LIN {X 0,Y 573.262,Z 307.702,A -85,B 0,C 180,E1 -2310.634,E2 -2310.634} C_VEL
LIN {X 0,Y 573.263,Z 307.696,A -85,B 0,C 180,E1 -2313.5,E2 -2313.5} C_VEL
LIN {X 0,Y 573.221,Z 307.71,A -85,B 0,C 180,E1 -2316.134,E2 -2316.134} C_VEL
LIN {X 0,Y 573.242,Z 307.699,A -85,B 0,C 180,E1 -2319.173,E2 -2319.173} C_VEL
LIN {X 0,Y 573.221,Z 307.701,A -85,B 0,C 180,E1 -2321.411,E2 -2321.411} C_VEL
LIN {X 0,Y 573.236,Z 307.703,A -85,B 0,C 180,E1 -2323.621,E2 -2323.621} C_VEL
LIN {X 0,Y 573.263,Z 307.702,A -85,B 0,C 180,E1 -2325.807,E2 -2325.807} C_VEL
LIN {X 0,Y 573.254,Z 307.697,A -85,B 0,C 180,E1 -2328.745,E2 -2328.745} C_VEL
LIN {X 0,Y 573.271,Z 307.7,A -85,B 0,C 180,E1 -2331.54,E2 -2331.54} C_VEL
LIN {X 0,Y 573.231,Z 307.706,A -85,B 0,C 180,E1 -2333.665,E2 -2333.665} C_VEL
LIN {X 0,Y 573.212,Z 307.713,A -85,B 0,C 180,E1 -2335.781,E2 -2335.781} C_VEL
LIN {X 0,Y 573.289,Z 307.701,A -85,B 0,C 180,E1 -2337.892,E2 -2337.892} C_VEL
LIN {X 0,Y 573.301,Z 307.696,A -85,B 0,C 180,E1 -2340,E2 -2340} C_VEL
LIN {X 0,Y 573.272,Z 307.695,A -85,B 0,C 180,E1 -2342.811,E2 -2342.811} C_VEL
LIN {X 0,Y 573.263,Z 307.705,A -85,B 0,C 180,E1 -2345.628,E2 -2345.628} C_VEL
LIN {X 0,Y 573.22,Z 307.701,A -85,B 0,C 180,E1 -2348.46,E2 -2348.46} C_VEL
LIN {X 0,Y 573.261,Z 307.704,A -85,B 0,C 180,E1 -2351.312,E2 -2351.312} C_VEL
LIN {X 0,Y 573.214,Z 307.703,A -85,B 0,C 180,E1 -2354.402,E2 -2354.402} C_VEL
LIN {X 0,Y 573.226,Z 307.706,A -85,B 0,C 180,E1 -2357.112,E2 -2357.112} C_VEL
LIN {X 0,Y 573.217,Z 307.703,A -85,B 0,C 180,E1 -2360.078,E2 -2360.078} C_VEL
LIN {X 0,Y 573.207,Z 307.703,A -85,B 0,C 180,E1 -2362.339,E2 -2362.339} C_VEL
LIN {X 0,Y 573.184,Z 307.706,A -85,B 0,C 180,E1 -2364.34,E2 -2364.34} C_VEL
LIN {X 0,Y 572.546,Z 307.793,A -85,B 0,C 180,E1 -2364.927,E2 -2364.927} C_VEL
LIN {X 0,Y 569.716,Z 308.148,A -85,B 0,C 180,E1 -2365.879,E2 -2365.879} C_VEL
LIN {X 0,Y 567.302,Z 308.45,A -85,B 0,C 180,E1 -2366.645,E2 -2366.645} C_VEL
LIN {X 0,Y 566.251,Z 308.577,A -85,B 0,C 180,E1 -2367.236,E2 -2367.236} C_VEL
LIN {X 0,Y 566.158,Z 308.585,A -85,B 0,C 180,E1 -2367.436,E2 -2367.436} C_VEL
LIN {X 0,Y 566.159,Z 308.583,A -85,B 0,C 180,E1 -2369.771,E2 -2369.771} C_VEL
LIN {X 0,Y 566.189,Z 308.58,A -85,B 0,C 180,E1 -2372.429,E2 -2372.429} C_VEL
LIN {X 0,Y 566.168,Z 308.591,A -85,B 0,C 180,E1 -2374.989,E2 -2374.989} C_VEL
LIN {X 0,Y 566.186,Z 308.581,A -85,B 0,C 180,E1 -2377.461,E2 -2377.461} C_VEL
LIN {X 0,Y 566.197,Z 308.578,A -85,B 0,C 180,E1 -2380.199,E2 -2380.199} C_VEL
LIN {X 0,Y 566.191,Z 308.584,A -85,B 0,C 180,E1 -2383.055,E2 -2383.055} C_VEL
LIN {X 0,Y 566.185,Z 308.579,A -85,B 0,C 180,E1 -2386.05,E2 -2386.05} C_VEL
LIN {X 0,Y 566.195,Z 308.582,A -85,B 0,C 180,E1 -2389.215,E2 -2389.215} C_VEL
LIN {X 0,Y 566.227,Z 308.615,A -85,B 0,C 180,E1 -2391.146,E2 -2391.146} C_VEL
LIN {X 0,Y 566.73,Z 313.138,A -85,B 0,C 180,E1 -2391.908,E2 -2391.908} C_VEL
LIN {X 0,Y 566.547,Z 330.448,A -85,B 0,C 180,E1 -2394.685,E2 -2394.685} C_VEL
LIN {X 0,Y 566.522,Z 332.949,A -85,B 0,C 180,E1 -2395.082,E2 -2395.082} C_VEL
LIN {X 0,Y 567.796,Z 340.155,A -85,B 0,C 180,E1 -2395.217,E2 -2395.217} C_VEL
LIN {X 0,Y 567.419,Z 469.812,A -85,B 0,C 180,E1 -2396.898,E2 -2396.898} C_VEL
LIN {X 0,Y 567.292,Z 484.271,A -85,B 0,C 180,E1 -2397.238,E2 -2397.238} C_VEL
LIN {X 0,Y 567.159,Z 497.173,A -85,B 0,C 180,E1 -2397.674,E2 -2397.674} C_VEL
LIN {X 0,Y 567.003,Z 509.326,A -85,B 0,C 180,E1 -2398.212,E2 -2398.212} C_VEL
LIN {X 0,Y 566.77,Z 521.671,A -85,B 0,C 180,E1 -2398.901,E2 -2398.901} C_VEL
LIN {X 0,Y 566.622,Z 533.823,A -85,B 0,C 180,E1 -2399.744,E2 -2399.744} C_VEL
LIN {X 0,Y 566.424,Z 545.722,A -85,B 0,C 180,E1 -2400.756,E2 -2400.756} C_VEL
LIN {X 0,Y 566.262,Z 556.36,A -85,B 0,C 180,E1 -2401.861,E2 -2401.861} C_VEL
LIN {X 0,Y 566.116,Z 565.674,A -85,B 0,C 180,E1 -2403.045,E2 -2403.045} C_VEL
LIN {X 0,Y 566.036,Z 573.388,A -85,B 0,C 180,E1 -2404.243,E2 -2404.243} C_VEL
LIN {X 0,Y 565.952,Z 579.581,A -85,B 0,C 180,E1 -2405.418,E2 -2405.418} C_VEL
LIN {X 0,Y 565.903,Z 585.24,A -85,B 0,C 180,E1 -2406.781,E2 -2406.781} C_VEL
LIN {X 0,Y 565.881,Z 589.422,A -85,B 0,C 180,E1 -2408.126,E2 -2408.126} C_VEL
LIN {X 0,Y 565.89,Z 591.214,A -85,B 0,C 180,E1 -2408.891,E2 -2408.891} C_VEL
LIN {X 0,Y 565.829,Z 593.598,A -85,B 0,C 180,E1 -2410.406,E2 -2410.406} C_VEL
LIN {X 0,Y 565.832,Z 594.477,A -85,B 0,C 180,E1 -2411.91,E2 -2411.91} C_VEL
LIN {X 0,Y 565.844,Z 593.899,A -85,B 0,C 180,E1 -2413.402,E2 -2413.402} C_VEL
LIN {X 0,Y 565.832,Z 591.855,A -85,B 0,C 180,E1 -2414.881,E2 -2414.881} C_VEL
LIN {X 0,Y 565.895,Z 588.343,A -85,B 0,C 180,E1 -2416.352,E2 -2416.352} C_VEL
LIN {X 0,Y 565.943,Z 583.303,A -85,B 0,C 180,E1 -2417.813,E2 -2417.813} C_VEL
LIN {X 0,Y 565.977,Z 578.3,A -85,B 0,C 180,E1 -2418.931,E2 -2418.931} C_VEL
LIN {X 0,Y 566.065,Z 571.431,A -85,B 0,C 180,E1 -2420.171,E2 -2420.171} C_VEL
LIN {X 0,Y 566.122,Z 562.799,A -85,B 0,C 180,E1 -2421.433,E2 -2421.433} C_VEL
LIN {X 0,Y 566.317,Z 553.789,A -85,B 0,C 180,E1 -2422.513,E2 -2422.513} C_VEL
LIN {X 0,Y 566.46,Z 542.97,A -85,B 0,C 180,E1 -2423.59,E2 -2423.59} C_VEL
LIN {X 0,Y 566.637,Z 532.033,A -85,B 0,C 180,E1 -2424.485,E2 -2424.485} C_VEL
LIN {X 0,Y 566.828,Z 520.066,A -85,B 0,C 180,E1 -2425.289,E2 -2425.289} C_VEL
LIN {X 0,Y 567.004,Z 508.63,A -85,B 0,C 180,E1 -2425.914,E2 -2425.914} C_VEL
LIN {X 0,Y 567.186,Z 495.217,A -85,B 0,C 180,E1 -2426.493,E2 -2426.493} C_VEL
LIN {X 0,Y 567.312,Z 481.204,A -85,B 0,C 180,E1 -2426.938,E2 -2426.938} C_VEL
LIN {X 0,Y 567.44,Z 467.65,A -85,B 0,C 180,E1 -2427.228,E2 -2427.228} C_VEL
LIN {X 0,Y 567.666,Z 339.011,A -85,B 0,C 180,E1 -2428.892,E2 -2428.892} C_VEL
LIN {X 0,Y 566.496,Z 332.857,A -85,B 0,C 180,E1 -2429.023,E2 -2429.023} C_VEL
LIN {X 0,Y 566.728,Z 315.639,A -85,B 0,C 180,E1 -2431.777,E2 -2431.777} C_VEL
LIN {X 0,Y 566.513,Z 310.212,A -85,B 0,C 180,E1 -2432.667,E2 -2432.667} C_VEL
LIN {X 0,Y 566.216,Z 308.583,A -85,B 0,C 180,E1 -2432.98,E2 -2432.98} C_VEL
LIN {X 0,Y 566.245,Z 308.577,A -85,B 0,C 180,E1 -2435.699,E2 -2435.699} C_VEL
LIN {X 0,Y 566.19,Z 308.579,A -85,B 0,C 180,E1 -2438.567,E2 -2438.567} C_VEL
LIN {X 0,Y 566.24,Z 308.578,A -85,B 0,C 180,E1 -2441.455,E2 -2441.455} C_VEL
LIN {X 0,Y 566.203,Z 308.576,A -85,B 0,C 180,E1 -2444.495,E2 -2444.495} C_VEL
LIN {X 0,Y 566.185,Z 308.586,A -85,B 0,C 180,E1 -2447.333,E2 -2447.333} C_VEL
LIN {X 0,Y 566.197,Z 308.58,A -85,B 0,C 180,E1 -2449.582,E2 -2449.582} C_VEL
LIN {X 0,Y 566.181,Z 308.579,A -85,B 0,C 180,E1 -2451.864,E2 -2451.864} C_VEL
LIN {X 0,Y 566.177,Z 308.588,A -85,B 0,C 180,E1 -2455.022,E2 -2455.022} C_VEL
LIN {X 0,Y 566.159,Z 308.586,A -85,B 0,C 180,E1 -2457.342,E2 -2457.342} C_VEL
LIN {X 0,Y 566.156,Z 308.582,A -85,B 0,C 180,E1 -2459.772,E2 -2459.772} C_VEL
LIN {X 0,Y 566.174,Z 308.581,A -85,B 0,C 180,E1 -2462.426,E2 -2462.426} C_VEL
LIN {X 0,Y 566.161,Z 308.59,A -85,B 0,C 180,E1 -2464.987,E2 -2464.987} C_VEL
LIN {X 0,Y 566.175,Z 308.581,A -85,B 0,C 180,E1 -2467.463,E2 -2467.463} C_VEL
LIN {X 0,Y 566.202,Z 308.577,A -85,B 0,C 180,E1 -2470.2,E2 -2470.2} C_VEL
LIN {X 0,Y 566.133,Z 308.59,A -85,B 0,C 180,E1 -2473.061,E2 -2473.061} C_VEL
LIN {X 0,Y 566.141,Z 308.584,A -85,B 0,C 180,E1 -2476.055,E2 -2476.055} C_VEL
LIN {X 0,Y 566.142,Z 308.59,A -85,B 0,C 180,E1 -2478.858,E2 -2478.858} C_VEL
LIN {X 0,Y 566.155,Z 308.582,A -85,B 0,C 180,E1 -2481.45,E2 -2481.45} C_VEL
LIN {X 0,Y 566.156,Z 308.582,A -85,B 0,C 180,E1 -2483.793,E2 -2483.793} C_VEL
LIN {X 0,Y 566.195,Z 308.582,A -85,B 0,C 180,E1 -2486.269,E2 -2486.269} C_VEL
LIN {X 0,Y 566.175,Z 308.583,A -85,B 0,C 180,E1 -2488.927,E2 -2488.927} C_VEL
LIN {X 0,Y 566.141,Z 308.585,A -85,B 0,C 180,E1 -2491.854,E2 -2491.854} C_VEL
LIN {X 0,Y 566.188,Z 308.584,A -85,B 0,C 180,E1 -2494.25,E2 -2494.25} C_VEL
LIN {X 0,Y 566.156,Z 308.586,A -85,B 0,C 180,E1 -2496.723,E2 -2496.723} C_VEL
LIN {X 0,Y 566.191,Z 308.579,A -85,B 0,C 180,E1 -2498.902,E2 -2498.902} C_VEL
LIN {X 0,Y 566.186,Z 308.578,A -85,B 0,C 180,E1 -2501.172,E2 -2501.172} C_VEL
LIN {X 0,Y 566.174,Z 308.588,A -85,B 0,C 180,E1 -2504.152,E2 -2504.152} C_VEL
LIN {X 0,Y 566.17,Z 308.587,A -85,B 0,C 180,E1 -2506.358,E2 -2506.358} C_VEL
LIN {X 0,Y 566.234,Z 308.572,A -85,B 0,C 180,E1 -2509.27,E2 -2509.27} C_VEL
LIN {X 0,Y 566.22,Z 308.583,A -85,B 0,C 180,E1 -2512.153,E2 -2512.153} C_VEL
LIN {X 0,Y 566.264,Z 308.568,A -85,B 0,C 180,E1 -2515.016,E2 -2515.016} C_VEL
LIN {X 0,Y 566.281,Z 308.573,A -85,B 0,C 180,E1 -2517.866,E2 -2517.866} C_VEL
LIN {X 0,Y 566.3,Z 308.564,A -85,B 0,C 180,E1 -2520.711,E2 -2520.711} C_VEL
LIN {X 0,Y 566.262,Z 308.568,A -85,B 0,C 180,E1 -2522.846,E2 -2522.846} C_VEL
LIN {X 0,Y 566.251,Z 308.576,A -85,B 0,C 180,E1 -2525.699,E2 -2525.699} C_VEL
LIN {X 0,Y 566.227,Z 308.573,A -85,B 0,C 180,E1 -2528.566,E2 -2528.566} C_VEL
LIN {X 0,Y 566.245,Z 308.575,A -85,B 0,C 180,E1 -2531.454,E2 -2531.454} C_VEL
LIN {X 0,Y 566.237,Z 308.572,A -85,B 0,C 180,E1 -2534.506,E2 -2534.506} C_VEL
LIN {X 0,Y 566.201,Z 308.58,A -85,B 0,C 180,E1 -2537.332,E2 -2537.332} C_VEL
LIN {X 0,Y 566.215,Z 308.575,A -85,B 0,C 180,E1 -2540.337,E2 -2540.337} C_VEL
LIN {X 0,Y 566.172,Z 308.584,A -85,B 0,C 180,E1 -2543.281,E2 -2543.281} C_VEL
LIN {X 0,Y 566.218,Z 308.581,A -85,B 0,C 180,E1 -2545.749,E2 -2545.749} C_VEL
LIN {X 0,Y 566.206,Z 308.576,A -85,B 0,C 180,E1 -2548.202,E2 -2548.202} C_VEL
LIN {X 0,Y 566.193,Z 308.581,A -85,B 0,C 180,E1 -2551.076,E2 -2551.076} C_VEL
LIN {X 0,Y 566.215,Z 308.579,A -85,B 0,C 180,E1 -2553.734,E2 -2553.734} C_VEL
LIN {X 0,Y 566.186,Z 308.578,A -85,B 0,C 180,E1 -2556.571,E2 -2556.571} C_VEL
LIN {X 0,Y 566.217,Z 308.578,A -85,B 0,C 180,E1 -2559.686,E2 -2559.686} C_VEL
LIN {X 0,Y 566.206,Z 308.579,A -85,B 0,C 180,E1 -2562.917,E2 -2562.917} C_VEL
LIN {X 0,Y 566.197,Z 308.577,A -85,B 0,C 180,E1 -2566.049,E2 -2566.049} C_VEL
LIN {X 0,Y 566.207,Z 308.585,A -85,B 0,C 180,E1 -2569.214,E2 -2569.214} C_VEL
LIN {X 0,Y 566.192,Z 308.579,A -85,B 0,C 180,E1 -2571.637,E2 -2571.637} C_VEL
LIN {X 0,Y 566.167,Z 308.581,A -85,B 0,C 180,E1 -2574.308,E2 -2574.308} C_VEL
LIN {X 0,Y 566.223,Z 308.581,A -85,B 0,C 180,E1 -2576.898,E2 -2576.898} C_VEL
LIN {X 0,Y 566.177,Z 308.585,A -85,B 0,C 180,E1 -2579.407,E2 -2579.407} C_VEL
LIN {X 0,Y 566.216,Z 308.578,A -85,B 0,C 180,E1 -2581.857,E2 -2581.857} C_VEL
LIN {X 0,Y 566.231,Z 308.617,A -85,B 0,C 180,E1 -2584.793,E2 -2584.793} C_VEL
LIN {X 0,Y 567.462,Z 314.904,A -85,B 0,C 180,E1 -2585.682,E2 -2585.682} C_VEL
LIN {X 0,Y 567.205,Z 336.056,A -85,B 0,C 180,E1 -2588.445,E2 -2588.445} C_VEL
LIN {X 0,Y 566.881,Z 358.65,A -85,B 0,C 180,E1 -2591.383,E2 -2591.383} C_VEL
LIN {X 0,Y 566.687,Z 371.393,A -85,B 0,C 180,E1 -2593.018,E2 -2593.018} C_VEL
LIN {X 0,Y 567.797,Z 378.785,A -85,B 0,C 180,E1 -2593.154,E2 -2593.154} C_VEL
LIN {X 0,Y 567.459,Z 509.858,A -85,B 0,C 180,E1 -2594.855,E2 -2594.855} C_VEL
LIN {X 0,Y 567.278,Z 524.474,A -85,B 0,C 180,E1 -2595.198,E2 -2595.198} C_VEL
LIN {X 0,Y 567.121,Z 538.824,A -85,B 0,C 180,E1 -2595.695,E2 -2595.695} C_VEL
LIN {X 0,Y 566.967,Z 551.631,A -85,B 0,C 180,E1 -2596.286,E2 -2596.286} C_VEL
LIN {X 0,Y 566.769,Z 564.094,A -85,B 0,C 180,E1 -2597.011,E2 -2597.011} C_VEL
LIN {X 0,Y 566.574,Z 576.636,A -85,B 0,C 180,E1 -2597.917,E2 -2597.917} C_VEL
LIN {X 0,Y 566.447,Z 587.313,A -85,B 0,C 180,E1 -2598.86,E2 -2598.86} C_VEL
LIN {X 0,Y 566.206,Z 597.847,A -85,B 0,C 180,E1 -2599.992,E2 -2599.992} C_VEL
LIN {X 0,Y 566.137,Z 606.169,A -85,B 0,C 180,E1 -2601.073,E2 -2601.073} C_VEL
LIN {X 0,Y 566.047,Z 614.124,A -85,B 0,C 180,E1 -2602.329,E2 -2602.329} C_VEL
LIN {X 0,Y 565.925,Z 620.525,A -85,B 0,C 180,E1 -2603.582,E2 -2603.582} C_VEL
LIN {X 0,Y 565.929,Z 624.959,A -85,B 0,C 180,E1 -2604.655,E2 -2604.655} C_VEL
LIN {X 0,Y 565.956,Z 628.441,A -85,B 0,C 180,E1 -2605.726,E2 -2605.726} C_VEL
LIN {X 0,Y 565.875,Z 631.831,A -85,B 0,C 180,E1 -2607.152,E2 -2607.152} C_VEL
LIN {X 0,Y 565.84,Z 633.832,A -85,B 0,C 180,E1 -2608.576,E2 -2608.576} C_VEL
LIN {X 0,Y 565.837,Z 634.5,A -85,B 0,C 180,E1 -2609.999,E2 -2609.999} C_VEL
LIN {X 0,Y 565.84,Z 633.835,A -85,B 0,C 180,E1 -2611.423,E2 -2611.423} C_VEL
LIN {X 0,Y 565.874,Z 631.835,A -85,B 0,C 180,E1 -2612.847,E2 -2612.847} C_VEL
LIN {X 0,Y 565.956,Z 628.447,A -85,B 0,C 180,E1 -2614.272,E2 -2614.272} C_VEL
LIN {X 0,Y 565.984,Z 623.571,A -85,B 0,C 180,E1 -2615.7,E2 -2615.7} C_VEL
LIN {X 0,Y 565.994,Z 619.048,A -85,B 0,C 180,E1 -2616.738,E2 -2616.738} C_VEL
LIN {X 0,Y 566.046,Z 612.041,A -85,B 0,C 180,E1 -2618.029,E2 -2618.029} C_VEL
LIN {X 0,Y 566.18,Z 603.563,A -85,B 0,C 180,E1 -2619.286,E2 -2619.286} C_VEL
LIN {X 0,Y 566.294,Z 594.714,A -85,B 0,C 180,E1 -2620.366,E2 -2620.366} C_VEL
LIN {X 0,Y 566.484,Z 583.997,A -85,B 0,C 180,E1 -2621.449,E2 -2621.449} C_VEL
LIN {X 0,Y 566.607,Z 573.149,A -85,B 0,C 180,E1 -2622.354,E2 -2622.354} C_VEL
LIN {X 0,Y 566.779,Z 561.267,A -85,B 0,C 180,E1 -2623.17,E2 -2623.17} C_VEL
LIN {X 0,Y 567.023,Z 548.111,A -85,B 0,C 180,E1 -2623.894,E2 -2623.894} C_VEL
LIN {X 0,Y 567.215,Z 535.047,A -85,B 0,C 180,E1 -2624.453,E2 -2624.453} C_VEL
LIN {X 0,Y 567.353,Z 521.152,A -85,B 0,C 180,E1 -2624.893,E2 -2624.893} C_VEL
LIN {X 0,Y 567.451,Z 507.181,A -85,B 0,C 180,E1 -2625.189,E2 -2625.189} C_VEL
LIN {X 0,Y 567.736,Z 377.314,A -85,B 0,C 180,E1 -2626.867,E2 -2626.867} C_VEL
LIN {X 0,Y 566.675,Z 371.403,A -85,B 0,C 180,E1 -2626.981,E2 -2626.981} C_VEL
LIN {X 0,Y 566.974,Z 350.117,A -85,B 0,C 180,E1 -2629.722,E2 -2629.722} C_VEL
LIN {X 0,Y 567.287,Z 329.609,A -85,B 0,C 180,E1 -2632.392,E2 -2632.392} C_VEL
LIN {X 0,Y 567.457,Z 314.872,A -85,B 0,C 180,E1 -2634.317,E2 -2634.317} C_VEL
LIN {X 0,Y 566.224,Z 308.582,A -85,B 0,C 180,E1 -2635.23,E2 -2635.23} C_VEL
LIN {X 0,Y 566.201,Z 308.579,A -85,B 0,C 180,E1 -2638.201,E2 -2638.201} C_VEL
LIN {X 0,Y 566.197,Z 308.585,A -85,B 0,C 180,E1 -2641.077,E2 -2641.077} C_VEL
LIN {X 0,Y 566.21,Z 308.575,A -85,B 0,C 180,E1 -2643.733,E2 -2643.733} C_VEL
LIN {X 0,Y 566.214,Z 308.58,A -85,B 0,C 180,E1 -2646.568,E2 -2646.568} C_VEL
LIN {X 0,Y 566.209,Z 308.576,A -85,B 0,C 180,E1 -2649.685,E2 -2649.685} C_VEL
LIN {X 0,Y 566.206,Z 308.576,A -85,B 0,C 180,E1 -2652.087,E2 -2652.087} C_VEL
LIN {X 0,Y 566.169,Z 308.583,A -85,B 0,C 180,E1 -2655.035,E2 -2655.035} C_VEL
LIN {X 0,Y 566.214,Z 308.578,A -85,B 0,C 180,E1 -2658.135,E2 -2658.135} C_VEL
LIN {X 0,Y 566.216,Z 308.58,A -85,B 0,C 180,E1 -2660.726,E2 -2660.726} C_VEL
LIN {X 0,Y 566.209,Z 308.576,A -85,B 0,C 180,E1 -2663.783,E2 -2663.783} C_VEL
LIN {X 0,Y 566.223,Z 308.576,A -85,B 0,C 180,E1 -2666.898,E2 -2666.898} C_VEL
LIN {X 0,Y 566.18,Z 308.579,A -85,B 0,C 180,E1 -2669.407,E2 -2669.407} C_VEL
LIN {X 0,Y 566.222,Z 308.577,A -85,B 0,C 180,E1 -2671.858,E2 -2671.858} C_VEL
LIN {X 0,Y 566.219,Z 308.582,A -85,B 0,C 180,E1 -2674.251,E2 -2674.251} C_VEL
LIN {X 0,Y 566.162,Z 308.582,A -85,B 0,C 180,E1 -2676.718,E2 -2676.718} C_VEL
LIN {X 0,Y 566.205,Z 308.579,A -85,B 0,C 180,E1 -2679.662,E2 -2679.662} C_VEL
LIN {X 0,Y 566.193,Z 308.579,A -85,B 0,C 180,E1 -2682.668,E2 -2682.668} C_VEL
LIN {X 0,Y 566.225,Z 308.576,A -85,B 0,C 180,E1 -2685.626,E2 -2685.626} C_VEL
LIN {X 0,Y 566.226,Z 308.572,A -85,B 0,C 180,E1 -2688.675,E2 -2688.675} C_VEL
LIN {X 0,Y 566.215,Z 308.577,A -85,B 0,C 180,E1 -2691.434,E2 -2691.434} C_VEL
LIN {X 0,Y 566.234,Z 308.575,A -85,B 0,C 180,E1 -2694.301,E2 -2694.301} C_VEL
LIN {X 0,Y 566.261,Z 308.577,A -85,B 0,C 180,E1 -2697.866,E2 -2697.866} C_VEL
LIN {X 0,Y 566.27,Z 308.572,A -85,B 0,C 180,E1 -2700,E2 -2700} C_VEL
LIN {X 0,Y 566.241,Z 308.571,A -85,B 0,C 180,E1 -2702.845,E2 -2702.845} C_VEL
LIN {X 0,Y 566.229,Z 308.581,A -85,B 0,C 180,E1 -2705.698,E2 -2705.698} C_VEL
LIN {X 0,Y 566.174,Z 308.579,A -85,B 0,C 180,E1 -2708.566,E2 -2708.566} C_VEL
LIN {X 0,Y 566.227,Z 308.583,A -85,B 0,C 180,E1 -2711.454,E2 -2711.454} C_VEL
LIN {X 0,Y 566.164,Z 308.581,A -85,B 0,C 180,E1 -2714.483,E2 -2714.483} C_VEL
LIN {X 0,Y 566.17,Z 308.589,A -85,B 0,C 180,E1 -2717.332,E2 -2717.332} C_VEL
LIN {X 0,Y 566.186,Z 308.584,A -85,B 0,C 180,E1 -2719.581,E2 -2719.581} C_VEL
LIN {X 0,Y 566.173,Z 308.58,A -85,B 0,C 180,E1 -2721.863,E2 -2721.863} C_VEL
LIN {X 0,Y 566.167,Z 308.588,A -85,B 0,C 180,E1 -2725.021,E2 -2725.021} C_VEL
LIN {X 0,Y 566.158,Z 308.585,A -85,B 0,C 180,E1 -2727.436,E2 -2727.436} C_VEL
LIN {X 0,Y 565.473,Z 308.668,A -85,B 0,C 180,E1 -2728.03,E2 -2728.03} C_VEL
LIN {X 0,Y 562.615,Z 309.029,A -85,B 0,C 180,E1 -2728.994,E2 -2728.994} C_VEL
LIN {X 0,Y 560.216,Z 309.324,A -85,B 0,C 180,E1 -2729.769,E2 -2729.769} C_VEL
LIN {X 0,Y 559.197,Z 309.451,A -85,B 0,C 180,E1 -2730.368,E2 -2730.368} C_VEL
LIN {X 0,Y 559.118,Z 309.462,A -85,B 0,C 180,E1 -2730.571,E2 -2730.571} C_VEL
LIN {X 0,Y 559.14,Z 309.461,A -85,B 0,C 180,E1 -2732.716,E2 -2732.716} C_VEL
LIN {X 0,Y 559.116,Z 309.464,A -85,B 0,C 180,E1 -2735.324,E2 -2735.324} C_VEL
LIN {X 0,Y 559.121,Z 309.459,A -85,B 0,C 180,E1 -2738.018,E2 -2738.018} C_VEL
LIN {X 0,Y 559.146,Z 309.464,A -85,B 0,C 180,E1 -2740.813,E2 -2740.813} C_VEL
LIN {X 0,Y 559.129,Z 309.458,A -85,B 0,C 180,E1 -2743.735,E2 -2743.735} C_VEL
LIN {X 0,Y 559.137,Z 309.465,A -85,B 0,C 180,E1 -2746.804,E2 -2746.804} C_VEL
LIN {X 0,Y 559.147,Z 309.461,A -85,B 0,C 180,E1 -2749.188,E2 -2749.188} C_VEL
LIN {X 0,Y 559.182,Z 309.484,A -85,B 0,C 180,E1 -2750.981,E2 -2750.981} C_VEL
LIN {X 0,Y 559.798,Z 314.265,A -85,B 0,C 180,E1 -2751.808,E2 -2751.808} C_VEL
LIN {X 0,Y 559.56,Z 332.795,A -85,B 0,C 180,E1 -2754.84,E2 -2754.84} C_VEL
LIN {X 0,Y 559.859,Z 334.574,A -85,B 0,C 180,E1 -2754.897,E2 -2754.897} C_VEL
LIN {X 0,Y 560.967,Z 340.274,A -85,B 0,C 180,E1 -2755.007,E2 -2755.007} C_VEL
LIN {X 0,Y 560.571,Z 469.915,A -85,B 0,C 180,E1 -2756.711,E2 -2756.711} C_VEL
LIN {X 0,Y 560.428,Z 484.37,A -85,B 0,C 180,E1 -2757.055,E2 -2757.055} C_VEL
LIN {X 0,Y 560.256,Z 497.766,A -85,B 0,C 180,E1 -2757.518,E2 -2757.518} C_VEL
LIN {X 0,Y 560.071,Z 510.322,A -85,B 0,C 180,E1 -2758.09,E2 -2758.09} C_VEL
LIN {X 0,Y 559.793,Z 522.907,A -85,B 0,C 180,E1 -2758.814,E2 -2758.814} C_VEL
LIN {X 0,Y 559.652,Z 534.479,A -85,B 0,C 180,E1 -2759.64,E2 -2759.64} C_VEL
LIN {X 0,Y 559.426,Z 546.262,A -85,B 0,C 180,E1 -2760.664,E2 -2760.664} C_VEL
LIN {X 0,Y 559.253,Z 556.449,A -85,B 0,C 180,E1 -2761.742,E2 -2761.742} C_VEL
LIN {X 0,Y 559.086,Z 565.411,A -85,B 0,C 180,E1 -2762.892,E2 -2762.892} C_VEL
LIN {X 0,Y 558.971,Z 573.109,A -85,B 0,C 180,E1 -2764.094,E2 -2764.094} C_VEL
LIN {X 0,Y 558.896,Z 578.835,A -85,B 0,C 180,E1 -2765.178,E2 -2765.178} C_VEL
LIN {X 0,Y 558.873,Z 583.571,A -85,B 0,C 180,E1 -2766.272,E2 -2766.272} C_VEL
LIN {X 0,Y 558.805,Z 587.643,A -85,B 0,C 180,E1 -2767.444,E2 -2767.444} C_VEL
LIN {X 0,Y 558.777,Z 590.725,A -85,B 0,C 180,E1 -2768.609,E2 -2768.609} C_VEL
LIN {X 0,Y 558.732,Z 593.334,A -85,B 0,C 180,E1 -2770.147,E2 -2770.147} C_VEL
LIN {X 0,Y 558.771,Z 594.065,A -85,B 0,C 180,E1 -2770.913,E2 -2770.913} C_VEL
LIN {X 0,Y 558.741,Z 594.422,A -85,B 0,C 180,E1 -2772.43,E2 -2772.43} C_VEL
LIN {X 0,Y 558.737,Z 593.34,A -85,B 0,C 180,E1 -2773.936,E2 -2773.936} C_VEL
LIN {X 0,Y 558.778,Z 590.824,A -85,B 0,C 180,E1 -2775.432,E2 -2775.432} C_VEL
LIN {X 0,Y 558.81,Z 586.813,A -85,B 0,C 180,E1 -2776.917,E2 -2776.917} C_VEL
LIN {X 0,Y 558.869,Z 582.758,A -85,B 0,C 180,E1 -2778.025,E2 -2778.025} C_VEL
LIN {X 0,Y 558.929,Z 577.75,A -85,B 0,C 180,E1 -2779.129,E2 -2779.129} C_VEL
LIN {X 0,Y 559.015,Z 570.59,A -85,B 0,C 180,E1 -2780.412,E2 -2780.412} C_VEL
LIN {X 0,Y 559.085,Z 563.138,A -85,B 0,C 180,E1 -2781.507,E2 -2781.507} C_VEL
LIN {X 0,Y 559.295,Z 554.197,A -85,B 0,C 180,E1 -2782.6,E2 -2782.6} C_VEL
LIN {X 0,Y 559.468,Z 543.454,A -85,B 0,C 180,E1 -2783.69,E2 -2783.69} C_VEL
LIN {X 0,Y 559.658,Z 532.616,A -85,B 0,C 180,E1 -2784.596,E2 -2784.596} C_VEL
LIN {X 0,Y 559.894,Z 520.778,A -85,B 0,C 180,E1 -2785.411,E2 -2785.411} C_VEL
LIN {X 0,Y 560.098,Z 507.727,A -85,B 0,C 180,E1 -2786.133,E2 -2786.133} C_VEL
LIN {X 0,Y 560.35,Z 493.914,A -85,B 0,C 180,E1 -2786.72,E2 -2786.72} C_VEL
LIN {X 0,Y 560.474,Z 480.264,A -85,B 0,C 180,E1 -2787.148,E2 -2787.148} C_VEL
LIN {X 0,Y 560.615,Z 466.096,A -85,B 0,C 180,E1 -2787.441,E2 -2787.441} C_VEL
LIN {X 0,Y 560.885,Z 339.994,A -85,B 0,C 180,E1 -2789.089,E2 -2789.089} C_VEL
LIN {X 0,Y 559.509,Z 332.893,A -85,B 0,C 180,E1 -2789.236,E2 -2789.236} C_VEL
LIN {X 0,Y 559.809,Z 316.079,A -85,B 0,C 180,E1 -2791.979,E2 -2791.979} C_VEL
LIN {X 0,Y 559.607,Z 311.813,A -85,B 0,C 180,E1 -2792.7,E2 -2792.7} C_VEL
LIN {X 0,Y 559.177,Z 309.461,A -85,B 0,C 180,E1 -2793.153,E2 -2793.153} C_VEL
LIN {X 0,Y 559.212,Z 309.453,A -85,B 0,C 180,E1 -2795.771,E2 -2795.771} C_VEL
LIN {X 0,Y 559.157,Z 309.456,A -85,B 0,C 180,E1 -2798.675,E2 -2798.675} C_VEL
LIN {X 0,Y 559.203,Z 309.453,A -85,B 0,C 180,E1 -2801.601,E2 -2801.601} C_VEL
LIN {X 0,Y 559.152,Z 309.455,A -85,B 0,C 180,E1 -2804.577,E2 -2804.577} C_VEL
LIN {X 0,Y 559.13,Z 309.461,A -85,B 0,C 180,E1 -2807.558,E2 -2807.558} C_VEL
LIN {X 0,Y 559.161,Z 309.454,A -85,B 0,C 180,E1 -2809.838,E2 -2809.838} C_VEL
LIN {X 0,Y 559.127,Z 309.457,A -85,B 0,C 180,E1 -2812.154,E2 -2812.154} C_VEL
LIN {X 0,Y 559.136,Z 309.464,A -85,B 0,C 180,E1 -2815.178,E2 -2815.178} C_VEL
LIN {X 0,Y 559.104,Z 309.461,A -85,B 0,C 180,E1 -2817.717,E2 -2817.717} C_VEL
LIN {X 0,Y 559.099,Z 309.461,A -85,B 0,C 180,E1 -2820.186,E2 -2820.186} C_VEL
LIN {X 0,Y 559.132,Z 309.462,A -85,B 0,C 180,E1 -2822.717,E2 -2822.717} C_VEL
LIN {X 0,Y 559.113,Z 309.462,A -85,B 0,C 180,E1 -2825.326,E2 -2825.326} C_VEL
LIN {X 0,Y 559.103,Z 309.46,A -85,B 0,C 180,E1 -2828.02,E2 -2828.02} C_VEL
LIN {X 0,Y 559.151,Z 309.454,A -85,B 0,C 180,E1 -2829.941,E2 -2829.941} C_VEL
LIN {X 0,Y 559.086,Z 309.466,A -85,B 0,C 180,E1 -2833.19,E2 -2833.19} C_VEL
LIN {X 0,Y 559.11,Z 309.459,A -85,B 0,C 180,E1 -2835.766,E2 -2835.766} C_VEL
LIN {X 0,Y 559.096,Z 309.464,A -85,B 0,C 180,E1 -2838.224,E2 -2838.224} C_VEL
LIN {X 0,Y 559.122,Z 309.461,A -85,B 0,C 180,E1 -2841.062,E2 -2841.062} C_VEL
LIN {X 0,Y 559.111,Z 309.459,A -85,B 0,C 180,E1 -2843.787,E2 -2843.787} C_VEL
LIN {X 0,Y 559.144,Z 309.463,A -85,B 0,C 180,E1 -2846.424,E2 -2846.424} C_VEL
LIN {X 0,Y 559.14,Z 309.458,A -85,B 0,C 180,E1 -2848.98,E2 -2848.98} C_VEL
LIN {X 0,Y 559.103,Z 309.46,A -85,B 0,C 180,E1 -2851.632,E2 -2851.632} C_VEL
LIN {X 0,Y 559.153,Z 309.456,A -85,B 0,C 180,E1 -2853.902,E2 -2853.902} C_VEL
LIN {X 0,Y 559.105,Z 309.466,A -85,B 0,C 180,E1 -2856.581,E2 -2856.581} C_VEL
LIN {X 0,Y 559.149,Z 309.454,A -85,B 0,C 180,E1 -2859.395,E2 -2859.395} C_VEL
LIN {X 0,Y 559.118,Z 309.46,A -85,B 0,C 180,E1 -2861.685,E2 -2861.685} C_VEL
LIN {X 0,Y 559.131,Z 309.46,A -85,B 0,C 180,E1 -2864.695,E2 -2864.695} C_VEL
LIN {X 0,Y 559.169,Z 309.454,A -85,B 0,C 180,E1 -2867.663,E2 -2867.663} C_VEL
LIN {X 0,Y 559.136,Z 309.461,A -85,B 0,C 180,E1 -2869.865,E2 -2869.865} C_VEL
LIN {X 0,Y 559.168,Z 309.453,A -85,B 0,C 180,E1 -2872.78,E2 -2872.78} C_VEL
LIN {X 0,Y 559.24,Z 309.443,A -85,B 0,C 180,E1 -2874.953,E2 -2874.953} C_VEL
LIN {X 0,Y 559.252,Z 309.448,A -85,B 0,C 180,E1 -2877.84,E2 -2877.84} C_VEL
LIN {X 0,Y 559.27,Z 309.44,A -85,B 0,C 180,E1 -2880.72,E2 -2880.72} C_VEL
LIN {X 0,Y 559.228,Z 309.445,A -85,B 0,C 180,E1 -2882.882,E2 -2882.882} C_VEL
LIN {X 0,Y 559.221,Z 309.453,A -85,B 0,C 180,E1 -2885.77,E2 -2885.77} C_VEL
LIN {X 0,Y 559.186,Z 309.45,A -85,B 0,C 180,E1 -2888.675,E2 -2888.675} C_VEL
LIN {X 0,Y 559.208,Z 309.454,A -85,B 0,C 180,E1 -2891.601,E2 -2891.601} C_VEL
LIN {X 0,Y 559.204,Z 309.448,A -85,B 0,C 180,E1 -2894.596,E2 -2894.596} C_VEL
LIN {X 0,Y 559.16,Z 309.461,A -85,B 0,C 180,E1 -2897.557,E2 -2897.557} C_VEL
LIN {X 0,Y 559.173,Z 309.458,A -85,B 0,C 180,E1 -2899.838,E2 -2899.838} C_VEL
LIN {X 0,Y 559.143,Z 309.457,A -85,B 0,C 180,E1 -2902.153,E2 -2902.153} C_VEL
LIN {X 0,Y 559.18,Z 309.456,A -85,B 0,C 180,E1 -2905.298,E2 -2905.298} C_VEL
LIN {X 0,Y 559.172,Z 309.452,A -85,B 0,C 180,E1 -2908.381,E2 -2908.381} C_VEL
LIN {X 0,Y 559.149,Z 309.461,A -85,B 0,C 180,E1 -2911.273,E2 -2911.273} C_VEL
LIN {X 0,Y 559.169,Z 309.454,A -85,B 0,C 180,E1 -2913.949,E2 -2913.949} C_VEL
LIN {X 0,Y 559.135,Z 309.462,A -85,B 0,C 180,E1 -2917.109,E2 -2917.109} C_VEL
LIN {X 0,Y 559.163,Z 309.454,A -85,B 0,C 180,E1 -2919.941,E2 -2919.941} C_VEL
LIN {X 0,Y 559.162,Z 309.455,A -85,B 0,C 180,E1 -2922.744,E2 -2922.744} C_VEL
LIN {X 0,Y 559.152,Z 309.456,A -85,B 0,C 180,E1 -2925.761,E2 -2925.761} C_VEL
LIN {X 0,Y 559.166,Z 309.452,A -85,B 0,C 180,E1 -2928.23,E2 -2928.23} C_VEL
LIN {X 0,Y 559.182,Z 309.459,A -85,B 0,C 180,E1 -2931.191,E2 -2931.191} C_VEL
LIN {X 0,Y 559.143,Z 309.456,A -85,B 0,C 180,E1 -2933.789,E2 -2933.789} C_VEL
LIN {X 0,Y 559.166,Z 309.454,A -85,B 0,C 180,E1 -2936.425,E2 -2936.425} C_VEL
LIN {X 0,Y 559.154,Z 309.464,A -85,B 0,C 180,E1 -2938.98,E2 -2938.98} C_VEL
LIN {X 0,Y 559.172,Z 309.457,A -85,B 0,C 180,E1 -2941.619,E2 -2941.619} C_VEL
LIN {X 0,Y 559.193,Z 309.51,A -85,B 0,C 180,E1 -2944.603,E2 -2944.603} C_VEL
LIN {X 0,Y 560.544,Z 316.14,A -85,B 0,C 180,E1 -2945.559,E2 -2945.559} C_VEL
LIN {X 0,Y 560.294,Z 335.79,A -85,B 0,C 180,E1 -2948.158,E2 -2948.158} C_VEL
LIN {X 0,Y 559.989,Z 357.202,A -85,B 0,C 180,E1 -2950.955,E2 -2950.955} C_VEL
LIN {X 0,Y 559.762,Z 371.378,A -85,B 0,C 180,E1 -2952.799,E2 -2952.799} C_VEL
LIN {X 0,Y 561.011,Z 379.047,A -85,B 0,C 180,E1 -2952.947,E2 -2952.947} C_VEL
LIN {X 0,Y 560.624,Z 508.599,A -85,B 0,C 180,E1 -2954.643,E2 -2954.643} C_VEL
LIN {X 0,Y 560.439,Z 523.048,A -85,B 0,C 180,E1 -2954.97,E2 -2954.97} C_VEL
LIN {X 0,Y 560.306,Z 536.493,A -85,B 0,C 180,E1 -2955.422,E2 -2955.422} C_VEL
LIN {X 0,Y 560.087,Z 549.865,A -85,B 0,C 180,E1 -2956.021,E2 -2956.021} C_VEL
LIN {X 0,Y 559.812,Z 562.668,A -85,B 0,C 180,E1 -2956.755,E2 -2956.755} C_VEL
LIN {X 0,Y 559.638,Z 574.304,A -85,B 0,C 180,E1 -2957.581,E2 -2957.581} C_VEL
LIN {X 0,Y 559.439,Z 584.878,A -85,B 0,C 180,E1 -2958.488,E2 -2958.488} C_VEL
LIN {X 0,Y 559.273,Z 594.701,A -85,B 0,C 180,E1 -2959.501,E2 -2959.501} C_VEL
LIN {X 0,Y 559.118,Z 603.553,A -85,B 0,C 180,E1 -2960.595,E2 -2960.595} C_VEL
LIN {X 0,Y 558.986,Z 612.032,A -85,B 0,C 180,E1 -2961.868,E2 -2961.868} C_VEL
LIN {X 0,Y 558.902,Z 618.863,A -85,B 0,C 180,E1 -2963.139,E2 -2963.139} C_VEL
LIN {X 0,Y 558.917,Z 623.566,A -85,B 0,C 180,E1 -2964.226,E2 -2964.226} C_VEL
LIN {X 0,Y 558.865,Z 628.442,A -85,B 0,C 180,E1 -2965.672,E2 -2965.672} C_VEL
LIN {X 0,Y 558.796,Z 631.831,A -85,B 0,C 180,E1 -2967.116,E2 -2967.116} C_VEL
LIN {X 0,Y 558.74,Z 633.833,A -85,B 0,C 180,E1 -2968.558,E2 -2968.558} C_VEL
LIN {X 0,Y 558.738,Z 634.5,A -85,B 0,C 180,E1 -2969.999,E2 -2969.999} C_VEL
LIN {X 0,Y 558.74,Z 633.835,A -85,B 0,C 180,E1 -2971.441,E2 -2971.441} C_VEL
LIN {X 0,Y 558.796,Z 631.836,A -85,B 0,C 180,E1 -2972.883,E2 -2972.883} C_VEL
LIN {X 0,Y 558.865,Z 628.448,A -85,B 0,C 180,E1 -2974.327,E2 -2974.327} C_VEL
LIN {X 0,Y 558.913,Z 623.571,A -85,B 0,C 180,E1 -2975.773,E2 -2975.773} C_VEL
LIN {X 0,Y 558.906,Z 617.057,A -85,B 0,C 180,E1 -2977.223,E2 -2977.223} C_VEL
LIN {X 0,Y 559.027,Z 609.806,A -85,B 0,C 180,E1 -2978.494,E2 -2978.494} C_VEL
LIN {X 0,Y 559.146,Z 600.828,A -85,B 0,C 180,E1 -2979.769,E2 -2979.769} C_VEL
LIN {X 0,Y 559.35,Z 591.399,A -85,B 0,C 180,E1 -2980.863,E2 -2980.863} C_VEL
LIN {X 0,Y 559.517,Z 580.962,A -85,B 0,C 180,E1 -2981.869,E2 -2981.869} C_VEL
LIN {X 0,Y 559.709,Z 569.443,A -85,B 0,C 180,E1 -2982.785,E2 -2982.785} C_VEL
LIN {X 0,Y 559.963,Z 556.654,A -85,B 0,C 180,E1 -2983.61,E2 -2983.61} C_VEL
LIN {X 0,Y 560.164,Z 544.165,A -85,B 0,C 180,E1 -2984.253,E2 -2984.253} C_VEL
LIN {X 0,Y 560.408,Z 531.097,A -85,B 0,C 180,E1 -2984.774,E2 -2984.774} C_VEL
LIN {X 0,Y 560.505,Z 517.564,A -85,B 0,C 180,E1 -2985.171,E2 -2985.171} C_VEL
LIN {X 0,Y 560.61,Z 502.658,A -85,B 0,C 180,E1 -2985.449,E2 -2985.449} C_VEL
LIN {X 0,Y 560.935,Z 378.12,A -85,B 0,C 180,E1 -2987.067,E2 -2987.067} C_VEL
LIN {X 0,Y 559.747,Z 371.371,A -85,B 0,C 180,E1 -2987.202,E2 -2987.202} C_VEL
LIN {X 0,Y 560.127,Z 348.478,A -85,B 0,C 180,E1 -2990.184,E2 -2990.184} C_VEL
LIN {X 0,Y 560.446,Z 324.932,A -85,B 0,C 180,E1 -2993.266,E2 -2993.266} C_VEL
LIN {X 0,Y 560.532,Z 316.096,A -85,B 0,C 180,E1 -2994.44,E2 -2994.44} C_VEL
LIN {X 0,Y 559.188,Z 309.458,A -85,B 0,C 180,E1 -2995.396,E2 -2995.396} C_VEL
LIN {X 0,Y 559.166,Z 309.456,A -85,B 0,C 180,E1 -2998.38,E2 -2998.38} C_VEL
LIN {X 0,Y 559.151,Z 309.46,A -85,B 0,C 180,E1 -3001.274,E2 -3001.274} C_VEL
LIN {X 0,Y 559.165,Z 309.452,A -85,B 0,C 180,E1 -3003.949,E2 -3003.949} C_VEL
LIN {X 0,Y 559.166,Z 309.456,A -85,B 0,C 180,E1 -3006.448,E2 -3006.448} C_VEL
LIN {X 0,Y 559.175,Z 309.459,A -85,B 0,C 180,E1 -3008.933,E2 -3008.933} C_VEL
LIN {X 0,Y 559.183,Z 309.45,A -85,B 0,C 180,E1 -3011.767,E2 -3011.767} C_VEL
LIN {X 0,Y 559.135,Z 309.463,A -85,B 0,C 180,E1 -3014.738,E2 -3014.738} C_VEL
LIN {X 0,Y 559.159,Z 309.455,A -85,B 0,C 180,E1 -3017.256,E2 -3017.256} C_VEL
LIN {X 0,Y 559.18,Z 309.453,A -85,B 0,C 180,E1 -3020.134,E2 -3020.134} C_VEL
LIN {X 0,Y 559.14,Z 309.46,A -85,B 0,C 180,E1 -3022.891,E2 -3022.891} C_VEL
LIN {X 0,Y 559.16,Z 309.457,A -85,B 0,C 180,E1 -3026.05,E2 -3026.05} C_VEL
LIN {X 0,Y 559.152,Z 309.456,A -85,B 0,C 180,E1 -3028.98,E2 -3028.98} C_VEL
LIN {X 0,Y 559.164,Z 309.454,A -85,B 0,C 180,E1 -3031.618,E2 -3031.618} C_VEL
LIN {X 0,Y 559.192,Z 309.453,A -85,B 0,C 180,E1 -3033.903,E2 -3033.903} C_VEL
LIN {X 0,Y 559.132,Z 309.46,A -85,B 0,C 180,E1 -3036.571,E2 -3036.571} C_VEL
LIN {X 0,Y 559.172,Z 309.453,A -85,B 0,C 180,E1 -3039.395,E2 -3039.395} C_VEL
LIN {X 0,Y 559.139,Z 309.458,A -85,B 0,C 180,E1 -3041.685,E2 -3041.685} C_VEL
LIN {X 0,Y 559.154,Z 309.462,A -85,B 0,C 180,E1 -3043.947,E2 -3043.947} C_VEL
LIN {X 0,Y 559.16,Z 309.461,A -85,B 0,C 180,E1 -3046.184,E2 -3046.184} C_VEL
LIN {X 0,Y 559.184,Z 309.449,A -85,B 0,C 180,E1 -3049.133,E2 -3049.133} C_VEL
LIN {X 0,Y 559.188,Z 309.455,A -85,B 0,C 180,E1 -3052.053,E2 -3052.053} C_VEL
LIN {X 0,Y 559.236,Z 309.444,A -85,B 0,C 180,E1 -3054.953,E2 -3054.953} C_VEL
LIN {X 0,Y 559.233,Z 309.453,A -85,B 0,C 180,E1 -3057.839,E2 -3057.839} C_VEL
LIN {X 0,Y 559.239,Z 309.448,A -85,B 0,C 180,E1 -3060,E2 -3060} C_VEL
LIN {X 0,Y 559.21,Z 309.448,A -85,B 0,C 180,E1 -3062.881,E2 -3062.881} C_VEL
LIN {X 0,Y 559.195,Z 309.456,A -85,B 0,C 180,E1 -3065.77,E2 -3065.77} C_VEL
LIN {X 0,Y 559.14,Z 309.455,A -85,B 0,C 180,E1 -3068.675,E2 -3068.675} C_VEL
LIN {X 0,Y 559.183,Z 309.457,A -85,B 0,C 180,E1 -3071.601,E2 -3071.601} C_VEL
LIN {X 0,Y 559.141,Z 309.456,A -85,B 0,C 180,E1 -3074.576,E2 -3074.576} C_VEL
LIN {X 0,Y 559.116,Z 309.465,A -85,B 0,C 180,E1 -3077.558,E2 -3077.558} C_VEL
LIN {X 0,Y 559.15,Z 309.457,A -85,B 0,C 180,E1 -3079.838,E2 -3079.838} C_VEL
LIN {X 0,Y 559.119,Z 309.458,A -85,B 0,C 180,E1 -3082.153,E2 -3082.153} C_VEL
LIN {X 0,Y 559.129,Z 309.466,A -85,B 0,C 180,E1 -3085.178,E2 -3085.178} C_VEL
LIN {X 0,Y 559.111,Z 309.46,A -85,B 0,C 180,E1 -3087.716,E2 -3087.716} C_VEL
LIN {X 0,Y 559.118,Z 309.462,A -85,B 0,C 180,E1 -3090.571,E2 -3090.571} C_VEL
LIN {X 0,Y 558.461,Z 309.55,A -85,B 0,C 180,E1 -3091.172,E2 -3091.172} C_VEL
LIN {X 0,Y 555.602,Z 309.906,A -85,B 0,C 180,E1 -3092.149,E2 -3092.149} C_VEL
LIN {X 0,Y 553.185,Z 310.205,A -85,B 0,C 180,E1 -3092.934,E2 -3092.934} C_VEL
LIN {X 0,Y 552.156,Z 310.329,A -85,B 0,C 180,E1 -3093.541,E2 -3093.541} C_VEL
LIN {X 0,Y 552.077,Z 310.337,A -85,B 0,C 180,E1 -3093.746,E2 -3093.746} C_VEL
LIN {X 0,Y 552.095,Z 310.34,A -85,B 0,C 180,E1 -3096.747,E2 -3096.747} C_VEL
LIN {X 0,Y 552.119,Z 310.332,A -85,B 0,C 180,E1 -3099.528,E2 -3099.528} C_VEL
LIN {X 0,Y 552.121,Z 310.333,A -85,B 0,C 180,E1 -3102.426,E2 -3102.426} C_VEL
LIN {X 0,Y 552.083,Z 310.336,A -85,B 0,C 180,E1 -3105.562,E2 -3105.562} C_VEL
LIN {X 0,Y 552.112,Z 310.34,A -85,B 0,C 180,E1 -3108.555,E2 -3108.555} C_VEL
LIN {X 0,Y 552.188,Z 310.499,A -85,B 0,C 180,E1 -3110.834,E2 -3110.834} C_VEL
LIN {X 0,Y 552.865,Z 315.939,A -85,B 0,C 180,E1 -3111.788,E2 -3111.788} C_VEL
LIN {X 0,Y 552.594,Z 332.988,A -85,B 0,C 180,E1 -3114.632,E2 -3114.632} C_VEL
LIN {X 0,Y 554.217,Z 342.155,A -85,B 0,C 180,E1 -3114.818,E2 -3114.818} C_VEL
LIN {X 0,Y 553.732,Z 469.915,A -85,B 0,C 180,E1 -3116.517,E2 -3116.517} C_VEL
LIN {X 0,Y 553.568,Z 484.62,A -85,B 0,C 180,E1 -3116.873,E2 -3116.873} C_VEL
LIN {X 0,Y 553.362,Z 499.061,A -85,B 0,C 180,E1 -3117.387,E2 -3117.387} C_VEL
LIN {X 0,Y 553.103,Z 512.319,A -85,B 0,C 180,E1 -3118.017,E2 -3118.017} C_VEL
LIN {X 0,Y 552.832,Z 525.266,A -85,B 0,C 180,E1 -3118.8,E2 -3118.8} C_VEL
LIN {X 0,Y 552.639,Z 537.064,A -85,B 0,C 180,E1 -3119.687,E2 -3119.687} C_VEL
LIN {X 0,Y 552.36,Z 547.821,A -85,B 0,C 180,E1 -3120.67,E2 -3120.67} C_VEL
LIN {X 0,Y 552.209,Z 557.6,A -85,B 0,C 180,E1 -3121.75,E2 -3121.75} C_VEL
LIN {X 0,Y 552.021,Z 566.33,A -85,B 0,C 180,E1 -3122.911,E2 -3122.911} C_VEL
LIN {X 0,Y 551.902,Z 573.941,A -85,B 0,C 180,E1 -3124.143,E2 -3124.143} C_VEL
LIN {X 0,Y 551.791,Z 580.902,A -85,B 0,C 180,E1 -3125.548,E2 -3125.548} C_VEL
LIN {X 0,Y 551.747,Z 585.57,A -85,B 0,C 180,E1 -3126.743,E2 -3126.743} C_VEL
LIN {X 0,Y 551.706,Z 589.185,A -85,B 0,C 180,E1 -3127.928,E2 -3127.928} C_VEL
LIN {X 0,Y 551.654,Z 591.793,A -85,B 0,C 180,E1 -3129.102,E2 -3129.102} C_VEL
LIN {X 0,Y 551.678,Z 593.904,A -85,B 0,C 180,E1 -3130.658,E2 -3130.658} C_VEL
LIN {X 0,Y 551.653,Z 594.474,A -85,B 0,C 180,E1 -3132.197,E2 -3132.197} C_VEL
LIN {X 0,Y 551.637,Z 593.599,A -85,B 0,C 180,E1 -3133.724,E2 -3133.724} C_VEL
LIN {X 0,Y 551.674,Z 591.291,A -85,B 0,C 180,E1 -3135.24,E2 -3135.24} C_VEL
LIN {X 0,Y 551.721,Z 587.523,A -85,B 0,C 180,E1 -3136.746,E2 -3136.746} C_VEL
LIN {X 0,Y 551.768,Z 583.664,A -85,B 0,C 180,E1 -3137.869,E2 -3137.869} C_VEL
LIN {X 0,Y 551.839,Z 578.895,A -85,B 0,C 180,E1 -3138.988,E2 -3138.988} C_VEL
LIN {X 0,Y 551.942,Z 571.994,A -85,B 0,C 180,E1 -3140.288,E2 -3140.288} C_VEL
LIN {X 0,Y 552.029,Z 563.482,A -85,B 0,C 180,E1 -3141.582,E2 -3141.582} C_VEL
LIN {X 0,Y 552.279,Z 554.604,A -85,B 0,C 180,E1 -3142.69,E2 -3142.69} C_VEL
LIN {X 0,Y 552.453,Z 543.946,A -85,B 0,C 180,E1 -3143.793,E2 -3143.793} C_VEL
LIN {X 0,Y 552.699,Z 532.042,A -85,B 0,C 180,E1 -3144.803,E2 -3144.803} C_VEL
LIN {X 0,Y 552.926,Z 520.089,A -85,B 0,C 180,E1 -3145.627,E2 -3145.627} C_VEL
LIN {X 0,Y 553.232,Z 506.742,A -85,B 0,C 180,E1 -3146.359,E2 -3146.359} C_VEL
LIN {X 0,Y 553.461,Z 493.913,A -85,B 0,C 180,E1 -3146.907,E2 -3146.907} C_VEL
LIN {X 0,Y 553.619,Z 480.236,A -85,B 0,C 180,E1 -3147.34,E2 -3147.34} C_VEL
LIN {X 0,Y 553.773,Z 466.046,A -85,B 0,C 180,E1 -3147.637,E2 -3147.637} C_VEL
LIN {X 0,Y 554.174,Z 341.276,A -85,B 0,C 180,E1 -3149.285,E2 -3149.285} C_VEL
LIN {X 0,Y 552.556,Z 333.017,A -85,B 0,C 180,E1 -3149.454,E2 -3149.454} C_VEL
LIN {X 0,Y 552.912,Z 315.518,A -85,B 0,C 180,E1 -3152.368,E2 -3152.368} C_VEL
LIN {X 0,Y 552.136,Z 310.338,A -85,B 0,C 180,E1 -3153.284,E2 -3153.284} C_VEL
LIN {X 0,Y 552.181,Z 310.328,A -85,B 0,C 180,E1 -3155.845,E2 -3155.845} C_VEL
LIN {X 0,Y 552.13,Z 310.333,A -85,B 0,C 180,E1 -3158.787,E2 -3158.787} C_VEL
LIN {X 0,Y 552.159,Z 310.328,A -85,B 0,C 180,E1 -3161.751,E2 -3161.751} C_VEL
LIN {X 0,Y 552.118,Z 310.333,A -85,B 0,C 180,E1 -3164.749,E2 -3164.749} C_VEL
LIN {X 0,Y 552.089,Z 310.336,A -85,B 0,C 180,E1 -3167.79,E2 -3167.79} C_VEL
LIN {X 0,Y 552.122,Z 310.33,A -85,B 0,C 180,E1 -3170.102,E2 -3170.102} C_VEL
LIN {X 0,Y 552.08,Z 310.336,A -85,B 0,C 180,E1 -3172.452,E2 -3172.452} C_VEL
LIN {X 0,Y 552.079,Z 310.341,A -85,B 0,C 180,E1 -3175.334,E2 -3175.334} C_VEL
LIN {X 0,Y 552.053,Z 310.338,A -85,B 0,C 180,E1 -3178.102,E2 -3178.102} C_VEL
LIN {X 0,Y 552.072,Z 310.34,A -85,B 0,C 180,E1 -3180.612,E2 -3180.612} C_VEL
LIN {X 0,Y 552.087,Z 310.34,A -85,B 0,C 180,E1 -3183.188,E2 -3183.188} C_VEL
LIN {X 0,Y 552.065,Z 310.337,A -85,B 0,C 180,E1 -3185.846,E2 -3185.846} C_VEL
LIN {X 0,Y 552.081,Z 310.34,A -85,B 0,C 180,E1 -3188.592,E2 -3188.592} C_VEL
LIN {X 0,Y 552.059,Z 310.34,A -85,B 0,C 180,E1 -3191.315,E2 -3191.315} C_VEL
LIN {X 0,Y 552.058,Z 310.339,A -85,B 0,C 180,E1 -3193.478,E2 -3193.478} C_VEL
LIN {X 0,Y 552.042,Z 310.347,A -85,B 0,C 180,E1 -3196.57,E2 -3196.57} C_VEL
LIN {X 0,Y 552.066,Z 310.337,A -85,B 0,C 180,E1 -3199.515,E2 -3199.515} C_VEL
LIN {X 0,Y 552.064,Z 310.342,A -85,B 0,C 180,E1 -3202.334,E2 -3202.334} C_VEL
LIN {X 0,Y 552.069,Z 310.339,A -85,B 0,C 180,E1 -3205.05,E2 -3205.05} C_VEL
LIN {X 0,Y 552.106,Z 310.332,A -85,B 0,C 180,E1 -3207.681,E2 -3207.681} C_VEL
LIN {X 0,Y 552.064,Z 310.342,A -85,B 0,C 180,E1 -3210.233,E2 -3210.233} C_VEL
LIN {X 0,Y 552.078,Z 310.337,A -85,B 0,C 180,E1 -3213.013,E2 -3213.013} C_VEL
LIN {X 0,Y 552.075,Z 310.339,A -85,B 0,C 180,E1 -3215.961,E2 -3215.961} C_VEL
LIN {X 0,Y 552.096,Z 310.333,A -85,B 0,C 180,E1 -3219.119,E2 -3219.119} C_VEL
LIN {X 0,Y 552.08,Z 310.335,A -85,B 0,C 180,E1 -3221.443,E2 -3221.443} C_VEL
LIN {X 0,Y 552.089,Z 310.34,A -85,B 0,C 180,E1 -3224.495,E2 -3224.495} C_VEL
LIN {X 0,Y 552.124,Z 310.33,A -85,B 0,C 180,E1 -3227.503,E2 -3227.503} C_VEL
LIN {X 0,Y 552.102,Z 310.335,A -85,B 0,C 180,E1 -3229.735,E2 -3229.735} C_VEL
LIN {X 0,Y 552.146,Z 310.334,A -85,B 0,C 180,E1 -3231.952,E2 -3231.952} C_VEL
LIN {X 0,Y 552.216,Z 310.318,A -85,B 0,C 180,E1 -3234.889,E2 -3234.889} C_VEL
LIN {X 0,Y 552.223,Z 310.323,A -85,B 0,C 180,E1 -3237.812,E2 -3237.812} C_VEL
LIN {X 0,Y 552.24,Z 310.316,A -85,B 0,C 180,E1 -3240.729,E2 -3240.729} C_VEL
LIN {X 0,Y 552.194,Z 310.321,A -85,B 0,C 180,E1 -3242.918,E2 -3242.918} C_VEL
LIN {X 0,Y 552.191,Z 310.33,A -85,B 0,C 180,E1 -3245.844,E2 -3245.844} C_VEL
LIN {X 0,Y 552.153,Z 310.326,A -85,B 0,C 180,E1 -3248.786,E2 -3248.786} C_VEL
LIN {X 0,Y 552.164,Z 310.334,A -85,B 0,C 180,E1 -3251.751,E2 -3251.751} C_VEL
LIN {X 0,Y 552.14,Z 310.328,A -85,B 0,C 180,E1 -3254.749,E2 -3254.749} C_VEL
LIN {X 0,Y 552.11,Z 310.339,A -85,B 0,C 180,E1 -3257.789,E2 -3257.789} C_VEL
LIN {X 0,Y 552.132,Z 310.332,A -85,B 0,C 180,E1 -3260.101,E2 -3260.101} C_VEL
LIN {X 0,Y 552.094,Z 310.333,A -85,B 0,C 180,E1 -3262.451,E2 -3262.451} C_VEL
LIN {X 0,Y 552.16,Z 310.331,A -85,B 0,C 180,E1 -3265.35,E2 -3265.35} C_VEL
LIN {X 0,Y 552.106,Z 310.333,A -85,B 0,C 180,E1 -3268.099,E2 -3268.099} C_VEL
LIN {X 0,Y 552.105,Z 310.332,A -85,B 0,C 180,E1 -3270.609,E2 -3270.609} C_VEL
LIN {X 0,Y 552.119,Z 310.336,A -85,B 0,C 180,E1 -3273.186,E2 -3273.186} C_VEL
LIN {X 0,Y 552.078,Z 310.338,A -85,B 0,C 180,E1 -3275.844,E2 -3275.844} C_VEL
LIN {X 0,Y 552.119,Z 310.331,A -85,B 0,C 180,E1 -3278.589,E2 -3278.589} C_VEL
LIN {X 0,Y 552.127,Z 310.336,A -85,B 0,C 180,E1 -3281.446,E2 -3281.446} C_VEL
LIN {X 0,Y 552.097,Z 310.334,A -85,B 0,C 180,E1 -3284.531,E2 -3284.531} C_VEL
LIN {X 0,Y 552.133,Z 310.332,A -85,B 0,C 180,E1 -3287.585,E2 -3287.585} C_VEL
LIN {X 0,Y 552.137,Z 310.329,A -85,B 0,C 180,E1 -3290.473,E2 -3290.473} C_VEL
LIN {X 0,Y 552.11,Z 310.337,A -85,B 0,C 180,E1 -3293.317,E2 -3293.317} C_VEL
LIN {X 0,Y 552.131,Z 310.329,A -85,B 0,C 180,E1 -3295.939,E2 -3295.939} C_VEL
LIN {X 0,Y 552.123,Z 310.334,A -85,B 0,C 180,E1 -3298.54,E2 -3298.54} C_VEL
LIN {X 0,Y 552.128,Z 310.336,A -85,B 0,C 180,E1 -3301.438,E2 -3301.438} C_VEL
LIN {X 0,Y 552.171,Z 310.355,A -85,B 0,C 180,E1 -3304.402,E2 -3304.402} C_VEL
LIN {X 0,Y 553.716,Z 318.862,A -85,B 0,C 180,E1 -3305.637,E2 -3305.637} C_VEL
LIN {X 0,Y 553.303,Z 340.904,A -85,B 0,C 180,E1 -3308.581,E2 -3308.581} C_VEL
LIN {X 0,Y 552.942,Z 362.91,A -85,B 0,C 180,E1 -3311.472,E2 -3311.472} C_VEL
LIN {X 0,Y 552.796,Z 371.441,A -85,B 0,C 180,E1 -3312.584,E2 -3312.584} C_VEL
LIN {X 0,Y 554.196,Z 379.266,A -85,B 0,C 180,E1 -3312.734,E2 -3312.734} C_VEL
LIN {X 0,Y 553.783,Z 509.857,A -85,B 0,C 180,E1 -3314.472,E2 -3314.472} C_VEL
LIN {X 0,Y 553.562,Z 524.266,A -85,B 0,C 180,E1 -3314.816,E2 -3314.816} C_VEL
LIN {X 0,Y 553.35,Z 538.821,A -85,B 0,C 180,E1 -3315.331,E2 -3315.331} C_VEL
LIN {X 0,Y 553.155,Z 551.628,A -85,B 0,C 180,E1 -3315.936,E2 -3315.936} C_VEL
LIN {X 0,Y 552.871,Z 564.091,A -85,B 0,C 180,E1 -3316.679,E2 -3316.679} C_VEL
LIN {X 0,Y 552.619,Z 576.64,A -85,B 0,C 180,E1 -3317.607,E2 -3317.607} C_VEL
LIN {X 0,Y 552.452,Z 587.269,A -85,B 0,C 180,E1 -3318.57,E2 -3318.57} C_VEL
LIN {X 0,Y 552.18,Z 597.848,A -85,B 0,C 180,E1 -3319.735,E2 -3319.735} C_VEL
LIN {X 0,Y 552.033,Z 606.171,A -85,B 0,C 180,E1 -3320.842,E2 -3320.842} C_VEL
LIN {X 0,Y 551.914,Z 614.124,A -85,B 0,C 180,E1 -3322.132,E2 -3322.132} C_VEL
LIN {X 0,Y 551.754,Z 620.803,A -85,B 0,C 180,E1 -3323.48,E2 -3323.48} C_VEL
LIN {X 0,Y 551.794,Z 624.959,A -85,B 0,C 180,E1 -3324.518,E2 -3324.518} C_VEL
LIN {X 0,Y 551.76,Z 628.442,A -85,B 0,C 180,E1 -3325.616,E2 -3325.616} C_VEL
LIN {X 0,Y 551.72,Z 631.831,A -85,B 0,C 180,E1 -3327.079,E2 -3327.079} C_VEL
LIN {X 0,Y 551.64,Z 633.833,A -85,B 0,C 180,E1 -3328.539,E2 -3328.539} C_VEL
LIN {X 0,Y 551.639,Z 634.5,A -85,B 0,C 180,E1 -3329.999,E2 -3329.999} C_VEL
LIN {X 0,Y 551.64,Z 633.836,A -85,B 0,C 180,E1 -3331.459,E2 -3331.459} C_VEL
LIN {X 0,Y 551.72,Z 631.836,A -85,B 0,C 180,E1 -3332.92,E2 -3332.92} C_VEL
LIN {X 0,Y 551.759,Z 628.449,A -85,B 0,C 180,E1 -3334.382,E2 -3334.382} C_VEL
LIN {X 0,Y 551.823,Z 623.57,A -85,B 0,C 180,E1 -3335.847,E2 -3335.847} C_VEL
LIN {X 0,Y 551.832,Z 617.058,A -85,B 0,C 180,E1 -3337.316,E2 -3337.316} C_VEL
LIN {X 0,Y 551.962,Z 609.807,A -85,B 0,C 180,E1 -3338.604,E2 -3338.604} C_VEL
LIN {X 0,Y 552.116,Z 600.828,A -85,B 0,C 180,E1 -3339.894,E2 -3339.894} C_VEL
LIN {X 0,Y 552.345,Z 591.4,A -85,B 0,C 180,E1 -3341.002,E2 -3341.002} C_VEL
LIN {X 0,Y 552.538,Z 580.962,A -85,B 0,C 180,E1 -3342.021,E2 -3342.021} C_VEL
LIN {X 0,Y 552.76,Z 569.44,A -85,B 0,C 180,E1 -3342.949,E2 -3342.949} C_VEL
LIN {X 0,Y 553.025,Z 556.653,A -85,B 0,C 180,E1 -3343.784,E2 -3343.784} C_VEL
LIN {X 0,Y 553.286,Z 544.163,A -85,B 0,C 180,E1 -3344.434,E2 -3344.434} C_VEL
LIN {X 0,Y 553.542,Z 530.968,A -85,B 0,C 180,E1 -3344.966,E2 -3344.966} C_VEL
LIN {X 0,Y 553.671,Z 517.426,A -85,B 0,C 180,E1 -3345.366,E2 -3345.366} C_VEL
LIN {X 0,Y 553.767,Z 502.658,A -85,B 0,C 180,E1 -3345.645,E2 -3345.645} C_VEL
LIN {X 0,Y 554.164,Z 379.133,A -85,B 0,C 180,E1 -3347.269,E2 -3347.269} C_VEL
LIN {X 0,Y 552.804,Z 371.355,A -85,B 0,C 180,E1 -3347.427,E2 -3347.427} C_VEL
LIN {X 0,Y 553.197,Z 348.223,A -85,B 0,C 180,E1 -3350.448,E2 -3350.448} C_VEL
LIN {X 0,Y 553.555,Z 324.755,A -85,B 0,C 180,E1 -3353.562,E2 -3353.562} C_VEL
LIN {X 0,Y 553.581,Z 317.332,A -85,B 0,C 180,E1 -3354.567,E2 -3354.567} C_VEL
LIN {X 0,Y 552.166,Z 310.332,A -85,B 0,C 180,E1 -3355.597,E2 -3355.597} C_VEL
LIN {X 0,Y 552.123,Z 310.336,A -85,B 0,C 180,E1 -3358.561,E2 -3358.561} C_VEL
LIN {X 0,Y 552.108,Z 310.335,A -85,B 0,C 180,E1 -3361.475,E2 -3361.475} C_VEL
LIN {X 0,Y 552.136,Z 310.329,A -85,B 0,C 180,E1 -3364.17,E2 -3364.17} C_VEL
LIN {X 0,Y 552.109,Z 310.339,A -85,B 0,C 180,E1 -3366.746,E2 -3366.746} C_VEL
LIN {X 0,Y 552.131,Z 310.33,A -85,B 0,C 180,E1 -3369.526,E2 -3369.526} C_VEL
LIN {X 0,Y 552.126,Z 310.333,A -85,B 0,C 180,E1 -3372.424,E2 -3372.424} C_VEL
LIN {X 0,Y 552.095,Z 310.331,A -85,B 0,C 180,E1 -3375.562,E2 -3375.562} C_VEL
LIN {X 0,Y 552.136,Z 310.335,A -85,B 0,C 180,E1 -3378.675,E2 -3378.675} C_VEL
LIN {X 0,Y 552.114,Z 310.33,A -85,B 0,C 180,E1 -3381.411,E2 -3381.411} C_VEL
LIN {X 0,Y 552.103,Z 310.337,A -85,B 0,C 180,E1 -3384.157,E2 -3384.157} C_VEL
LIN {X 0,Y 552.117,Z 310.334,A -85,B 0,C 180,E1 -3386.814,E2 -3386.814} C_VEL
LIN {X 0,Y 552.135,Z 310.332,A -85,B 0,C 180,E1 -3389.944,E2 -3389.944} C_VEL
LIN {X 0,Y 552.14,Z 310.328,A -85,B 0,C 180,E1 -3392.997,E2 -3392.997} C_VEL
LIN {X 0,Y 552.106,Z 310.332,A -85,B 0,C 180,E1 -3395.161,E2 -3395.161} C_VEL
LIN {X 0,Y 552.118,Z 310.338,A -85,B 0,C 180,E1 -3398.337,E2 -3398.337} C_VEL
LIN {X 0,Y 552.144,Z 310.328,A -85,B 0,C 180,E1 -3400.674,E2 -3400.674} C_VEL
LIN {X 0,Y 552.105,Z 310.337,A -85,B 0,C 180,E1 -3403.737,E2 -3403.737} C_VEL
LIN {X 0,Y 552.125,Z 310.338,A -85,B 0,C 180,E1 -3406.004,E2 -3406.004} C_VEL
LIN {X 0,Y 552.152,Z 310.324,A -85,B 0,C 180,E1 -3408.993,E2 -3408.993} C_VEL
LIN {X 0,Y 552.143,Z 310.335,A -85,B 0,C 180,E1 -3411.951,E2 -3411.951} C_VEL
LIN {X 0,Y 552.211,Z 310.319,A -85,B 0,C 180,E1 -3414.889,E2 -3414.889} C_VEL
LIN {X 0,Y 552.206,Z 310.328,A -85,B 0,C 180,E1 -3417.812,E2 -3417.812} C_VEL
LIN {X 0,Y 552.208,Z 310.324,A -85,B 0,C 180,E1 -3420,E2 -3420} C_VEL
LIN {X 0,Y 552.179,Z 310.324,A -85,B 0,C 180,E1 -3422.918,E2 -3422.918} C_VEL
LIN {X 0,Y 552.163,Z 310.331,A -85,B 0,C 180,E1 -3425.844,E2 -3425.844} C_VEL
LIN {X 0,Y 552.114,Z 310.331,A -85,B 0,C 180,E1 -3428.786,E2 -3428.786} C_VEL
LIN {X 0,Y 552.137,Z 310.332,A -85,B 0,C 180,E1 -3431.751,E2 -3431.751} C_VEL
LIN {X 0,Y 552.108,Z 310.333,A -85,B 0,C 180,E1 -3434.749,E2 -3434.749} C_VEL
LIN {X 0,Y 552.074,Z 310.339,A -85,B 0,C 180,E1 -3437.789,E2 -3437.789} C_VEL
LIN {X 0,Y 552.111,Z 310.332,A -85,B 0,C 180,E1 -3440.102,E2 -3440.102} C_VEL
LIN {X 0,Y 552.071,Z 310.336,A -85,B 0,C 180,E1 -3442.452,E2 -3442.452} C_VEL
LIN {X 0,Y 552.096,Z 310.337,A -85,B 0,C 180,E1 -3445.646,E2 -3445.646} C_VEL
LIN {X 0,Y 552.053,Z 310.337,A -85,B 0,C 180,E1 -3448.101,E2 -3448.101} C_VEL
LIN {X 0,Y 552.083,Z 310.339,A -85,B 0,C 180,E1 -3450.61,E2 -3450.61} C_VEL
LIN {X 0,Y 552.095,Z 310.341,A -85,B 0,C 180,E1 -3453.187,E2 -3453.187} C_VEL
LIN {X 0,Y 552.077,Z 310.337,A -85,B 0,C 180,E1 -3453.746,E2 -3453.746} C_VEL
LIN {X 0,Y 551.436,Z 310.419,A -85,B 0,C 180,E1 -3454.355,E2 -3454.355} C_VEL
LIN {X 0,Y 548.627,Z 310.772,A -85,B 0,C 180,E1 -3455.344,E2 -3455.344} C_VEL
LIN {X 0,Y 546.222,Z 311.075,A -85,B 0,C 180,E1 -3456.139,E2 -3456.139} C_VEL
LIN {X 0,Y 545.159,Z 311.206,A -85,B 0,C 180,E1 -3456.753,E2 -3456.753} C_VEL
LIN {X 0,Y 545.056,Z 311.217,A -85,B 0,C 180,E1 -3456.961,E2 -3456.961} C_VEL
LIN {X 0,Y 545.056,Z 311.211,A -85,B 0,C 180,E1 -3460.143,E2 -3460.143} C_VEL
LIN {X 0,Y 545.069,Z 311.214,A -85,B 0,C 180,E1 -3463.107,E2 -3463.107} C_VEL
LIN {X 0,Y 545.04,Z 311.215,A -85,B 0,C 180,E1 -3466.227,E2 -3466.227} C_VEL
LIN {X 0,Y 545.073,Z 311.217,A -85,B 0,C 180,E1 -3468.886,E2 -3468.886} C_VEL
LIN {X 0,Y 545.114,Z 311.213,A -85,B 0,C 180,E1 -3470.625,E2 -3470.625} C_VEL
LIN {X 0,Y 545.956,Z 317.476,A -85,B 0,C 180,E1 -3471.743,E2 -3471.743} C_VEL
LIN {X 0,Y 545.635,Z 333.283,A -85,B 0,C 180,E1 -3474.412,E2 -3474.412} C_VEL
LIN {X 0,Y 547.452,Z 342.839,A -85,B 0,C 180,E1 -3474.604,E2 -3474.604} C_VEL
LIN {X 0,Y 546.911,Z 470.102,A -85,B 0,C 180,E1 -3476.32,E2 -3476.32} C_VEL
LIN {X 0,Y 546.709,Z 484.655,A -85,B 0,C 180,E1 -3476.676,E2 -3476.676} C_VEL
LIN {X 0,Y 546.517,Z 498.356,A -85,B 0,C 180,E1 -3477.166,E2 -3477.166} C_VEL
LIN {X 0,Y 546.248,Z 510.362,A -85,B 0,C 180,E1 -3477.73,E2 -3477.73} C_VEL
LIN {X 0,Y 545.932,Z 522.849,A -85,B 0,C 180,E1 -3478.469,E2 -3478.469} C_VEL
LIN {X 0,Y 545.689,Z 535.074,A -85,B 0,C 180,E1 -3479.365,E2 -3479.365} C_VEL
LIN {X 0,Y 545.459,Z 546.26,A -85,B 0,C 180,E1 -3480.368,E2 -3480.368} C_VEL
LIN {X 0,Y 545.188,Z 556.786,A -85,B 0,C 180,E1 -3481.514,E2 -3481.514} C_VEL
LIN {X 0,Y 544.986,Z 565.268,A -85,B 0,C 180,E1 -3482.632,E2 -3482.632} C_VEL
LIN {X 0,Y 544.834,Z 573.661,A -85,B 0,C 180,E1 -3483.988,E2 -3483.988} C_VEL
LIN {X 0,Y 544.725,Z 579.802,A -85,B 0,C 180,E1 -3485.21,E2 -3485.21} C_VEL
LIN {X 0,Y 544.706,Z 584.726,A -85,B 0,C 180,E1 -3486.424,E2 -3486.424} C_VEL
LIN {X 0,Y 544.614,Z 588.506,A -85,B 0,C 180,E1 -3487.625,E2 -3487.625} C_VEL
LIN {X 0,Y 544.585,Z 591.312,A -85,B 0,C 180,E1 -3488.818,E2 -3488.818} C_VEL
LIN {X 0,Y 544.578,Z 593.665,A -85,B 0,C 180,E1 -3490.405,E2 -3490.405} C_VEL
LIN {X 0,Y 544.547,Z 594.488,A -85,B 0,C 180,E1 -3491.957,E2 -3491.957} C_VEL
LIN {X 0,Y 544.557,Z 593.853,A -85,B 0,C 180,E1 -3493.506,E2 -3493.506} C_VEL
LIN {X 0,Y 544.553,Z 591.759,A -85,B 0,C 180,E1 -3495.042,E2 -3495.042} C_VEL
LIN {X 0,Y 544.643,Z 588.201,A -85,B 0,C 180,E1 -3496.57,E2 -3496.57} C_VEL
LIN {X 0,Y 544.704,Z 583.119,A -85,B 0,C 180,E1 -3498.087,E2 -3498.087} C_VEL
LIN {X 0,Y 544.754,Z 578.212,A -85,B 0,C 180,E1 -3499.219,E2 -3499.219} C_VEL
LIN {X 0,Y 544.878,Z 571.156,A -85,B 0,C 180,E1 -3500.535,E2 -3500.535} C_VEL
LIN {X 0,Y 545.056,Z 562.458,A -85,B 0,C 180,E1 -3501.847,E2 -3501.847} C_VEL
LIN {X 0,Y 545.3,Z 552.664,A -85,B 0,C 180,E1 -3503.052,E2 -3503.052} C_VEL
LIN {X 0,Y 545.508,Z 541.476,A -85,B 0,C 180,E1 -3504.178,E2 -3504.178} C_VEL
LIN {X 0,Y 545.72,Z 530.218,A -85,B 0,C 180,E1 -3505.106,E2 -3505.106} C_VEL
LIN {X 0,Y 546.053,Z 517.781,A -85,B 0,C 180,E1 -3505.941,E2 -3505.941} C_VEL
LIN {X 0,Y 546.361,Z 505.808,A -85,B 0,C 180,E1 -3506.59,E2 -3506.59} C_VEL
LIN {X 0,Y 546.605,Z 492.712,A -85,B 0,C 180,E1 -3507.145,E2 -3507.145} C_VEL
LIN {X 0,Y 546.841,Z 478.454,A -85,B 0,C 180,E1 -3507.584,E2 -3507.584} C_VEL
LIN {X 0,Y 546.953,Z 464.613,A -85,B 0,C 180,E1 -3507.861,E2 -3507.861} C_VEL
LIN {X 0,Y 547.406,Z 342.21,A -85,B 0,C 180,E1 -3509.495,E2 -3509.495} C_VEL
LIN {X 0,Y 545.632,Z 333.155,A -85,B 0,C 180,E1 -3509.698,E2 -3509.698} C_VEL
LIN {X 0,Y 545.96,Z 316.049,A -85,B 0,C 180,E1 -3512.583,E2 -3512.583} C_VEL
LIN {X 0,Y 545.083,Z 311.217,A -85,B 0,C 180,E1 -3513.466,E2 -3513.466} C_VEL
LIN {X 0,Y 545.13,Z 311.206,A -85,B 0,C 180,E1 -3515.921,E2 -3515.921} C_VEL
LIN {X 0,Y 545.09,Z 311.209,A -85,B 0,C 180,E1 -3518.154,E2 -3518.154} C_VEL
LIN {X 0,Y 545.132,Z 311.206,A -85,B 0,C 180,E1 -3521.534,E2 -3521.534} C_VEL
LIN {X 0,Y 545.075,Z 311.212,A -85,B 0,C 180,E1 -3524.944,E2 -3524.944} C_VEL
LIN {X 0,Y 545.055,Z 311.21,A -85,B 0,C 180,E1 -3528.027,E2 -3528.027} C_VEL
LIN {X 0,Y 545.088,Z 311.206,A -85,B 0,C 180,E1 -3530.373,E2 -3530.373} C_VEL
LIN {X 0,Y 545.067,Z 311.211,A -85,B 0,C 180,E1 -3533.56,E2 -3533.56} C_VEL
LIN {X 0,Y 545.036,Z 311.212,A -85,B 0,C 180,E1 -3536.003,E2 -3536.003} C_VEL
LIN {X 0,Y 545.023,Z 311.219,A -85,B 0,C 180,E1 -3538.736,E2 -3538.736} C_VEL
LIN {X 0,Y 545.041,Z 311.213,A -85,B 0,C 180,E1 -3541.677,E2 -3541.677} C_VEL
LIN {X 0,Y 545.04,Z 311.216,A -85,B 0,C 180,E1 -3544.567,E2 -3544.567} C_VEL
LIN {X 0,Y 545.002,Z 311.22,A -85,B 0,C 180,E1 -3547.307,E2 -3547.307} C_VEL
LIN {X 0,Y 545.051,Z 311.212,A -85,B 0,C 180,E1 -3550.144,E2 -3550.144} C_VEL
LIN {X 0,Y 544.996,Z 311.222,A -85,B 0,C 180,E1 -3553.115,E2 -3553.115} C_VEL
LIN {X 0,Y 545.021,Z 311.217,A -85,B 0,C 180,E1 -3556.23,E2 -3556.23} C_VEL
LIN {X 0,Y 545.002,Z 311.223,A -85,B 0,C 180,E1 -3558.879,E2 -3558.879} C_VEL
LIN {X 0,Y 545.018,Z 311.215,A -85,B 0,C 180,E1 -3561.869,E2 -3561.869} C_VEL
LIN {X 0,Y 545.02,Z 311.223,A -85,B 0,C 180,E1 -3564.531,E2 -3564.531} C_VEL
LIN {X 0,Y 545.06,Z 311.211,A -85,B 0,C 180,E1 -3567.211,E2 -3567.211} C_VEL
LIN {X 0,Y 545.019,Z 311.215,A -85,B 0,C 180,E1 -3569.808,E2 -3569.808} C_VEL
LIN {X 0,Y 545.024,Z 311.218,A -85,B 0,C 180,E1 -3572.842,E2 -3572.842} C_VEL
LIN {X 0,Y 545.018,Z 311.215,A -85,B 0,C 180,E1 -3575.63,E2 -3575.63} C_VEL
LIN {X 0,Y 545.035,Z 311.215,A -85,B 0,C 180,E1 -3578.836,E2 -3578.836} C_VEL
LIN {X 0,Y 545.043,Z 311.212,A -85,B 0,C 180,E1 -3581.195,E2 -3581.195} C_VEL
LIN {X 0,Y 545.035,Z 311.222,A -85,B 0,C 180,E1 -3584.289,E2 -3584.289} C_VEL
LIN {X 0,Y 545.054,Z 311.214,A -85,B 0,C 180,E1 -3586.58,E2 -3586.58} C_VEL
LIN {X 0,Y 545.118,Z 311.203,A -85,B 0,C 180,E1 -3588.85,E2 -3588.85} C_VEL
LIN {X 0,Y 545.095,Z 311.21,A -85,B 0,C 180,E1 -3591.847,E2 -3591.847} C_VEL
LIN {X 0,Y 545.193,Z 311.194,A -85,B 0,C 180,E1 -3594.823,E2 -3594.823} C_VEL
LIN {X 0,Y 545.195,Z 311.198,A -85,B 0,C 180,E1 -3597.784,E2 -3597.784} C_VEL
LIN {X 0,Y 545.211,Z 311.191,A -85,B 0,C 180,E1 -3600.739,E2 -3600.739} C_VEL
LIN {X 0,Y 545.16,Z 311.197,A -85,B 0,C 180,E1 -3602.956,E2 -3602.956} C_VEL
LIN {X 0,Y 545.163,Z 311.206,A -85,B 0,C 180,E1 -3605.92,E2 -3605.92} C_VEL
LIN {X 0,Y 545.111,Z 311.203,A -85,B 0,C 180,E1 -3608.9,E2 -3608.9} C_VEL
LIN {X 0,Y 545.108,Z 311.211,A -85,B 0,C 180,E1 -3611.905,E2 -3611.905} C_VEL
LIN {X 0,Y 545.089,Z 311.206,A -85,B 0,C 180,E1 -3614.944,E2 -3614.944} C_VEL
LIN {X 0,Y 545.078,Z 311.212,A -85,B 0,C 180,E1 -3618.026,E2 -3618.026} C_VEL
LIN {X 0,Y 545.097,Z 311.206,A -85,B 0,C 180,E1 -3620.372,E2 -3620.372} C_VEL
LIN {X 0,Y 545.082,Z 311.216,A -85,B 0,C 180,E1 -3623.559,E2 -3623.559} C_VEL
LIN {X 0,Y 545.082,Z 311.21,A -85,B 0,C 180,E1 -3626.001,E2 -3626.001} C_VEL
LIN {X 0,Y 545.093,Z 311.206,A -85,B 0,C 180,E1 -3628.748,E2 -3628.748} C_VEL
LIN {X 0,Y 545.061,Z 311.215,A -85,B 0,C 180,E1 -3631.679,E2 -3631.679} C_VEL
LIN {X 0,Y 545.065,Z 311.209,A -85,B 0,C 180,E1 -3634.564,E2 -3634.564} C_VEL
LIN {X 0,Y 545.035,Z 311.221,A -85,B 0,C 180,E1 -3637.304,E2 -3637.304} C_VEL
LIN {X 0,Y 545.069,Z 311.209,A -85,B 0,C 180,E1 -3640.143,E2 -3640.143} C_VEL
LIN {X 0,Y 545.083,Z 311.214,A -85,B 0,C 180,E1 -3643.106,E2 -3643.106} C_VEL
LIN {X 0,Y 545.053,Z 311.21,A -85,B 0,C 180,E1 -3646.226,E2 -3646.226} C_VEL
LIN {X 0,Y 545.085,Z 311.211,A -85,B 0,C 180,E1 -3648.885,E2 -3648.885} C_VEL
LIN {X 0,Y 545.087,Z 311.211,A -85,B 0,C 180,E1 -3650.818,E2 -3650.818} C_VEL
LIN {X 0,Y 545.046,Z 311.213,A -85,B 0,C 180,E1 -3653.619,E2 -3653.619} C_VEL
LIN {X 0,Y 545.069,Z 311.209,A -85,B 0,C 180,E1 -3656.328,E2 -3656.328} C_VEL
LIN {X 0,Y 545.068,Z 311.219,A -85,B 0,C 180,E1 -3658.952,E2 -3658.952} C_VEL
LIN {X 0,Y 545.105,Z 311.211,A -85,B 0,C 180,E1 -3661.507,E2 -3661.507} C_VEL
LIN {X 0,Y 545.121,Z 311.273,A -85,B 0,C 180,E1 -3664.204,E2 -3664.204} C_VEL
LIN {X 0,Y 546.838,Z 320.122,A -85,B 0,C 180,E1 -3665.513,E2 -3665.513} C_VEL
LIN {X 0,Y 546.379,Z 342.142,A -85,B 0,C 180,E1 -3668.494,E2 -3668.494} C_VEL
LIN {X 0,Y 545.97,Z 364.147,A -85,B 0,C 180,E1 -3671.422,E2 -3671.422} C_VEL
LIN {X 0,Y 545.838,Z 371.198,A -85,B 0,C 180,E1 -3672.352,E2 -3672.352} C_VEL
LIN {X 0,Y 547.421,Z 380.603,A -85,B 0,C 180,E1 -3672.535,E2 -3672.535} C_VEL
LIN {X 0,Y 546.958,Z 509.821,A -85,B 0,C 180,E1 -3674.273,E2 -3674.273} C_VEL
LIN {X 0,Y 546.708,Z 524.417,A -85,B 0,C 180,E1 -3674.626,E2 -3674.626} C_VEL
LIN {X 0,Y 546.5,Z 538.82,A -85,B 0,C 180,E1 -3675.143,E2 -3675.143} C_VEL
LIN {X 0,Y 546.251,Z 551.626,A -85,B 0,C 180,E1 -3675.755,E2 -3675.755} C_VEL
LIN {X 0,Y 545.921,Z 564.089,A -85,B 0,C 180,E1 -3676.506,E2 -3676.506} C_VEL
LIN {X 0,Y 545.663,Z 576.642,A -85,B 0,C 180,E1 -3677.446,E2 -3677.446} C_VEL
LIN {X 0,Y 545.434,Z 587.832,A -85,B 0,C 180,E1 -3678.48,E2 -3678.48} C_VEL
LIN {X 0,Y 545.176,Z 597.847,A -85,B 0,C 180,E1 -3679.602,E2 -3679.602} C_VEL
LIN {X 0,Y 544.999,Z 606.17,A -85,B 0,C 180,E1 -3680.723,E2 -3680.723} C_VEL
LIN {X 0,Y 544.834,Z 614.123,A -85,B 0,C 180,E1 -3682.029,E2 -3682.029} C_VEL
LIN {X 0,Y 544.681,Z 621.165,A -85,B 0,C 180,E1 -3683.478,E2 -3683.478} C_VEL
LIN {X 0,Y 544.646,Z 626.199,A -85,B 0,C 180,E1 -3684.817,E2 -3684.817} C_VEL
LIN {X 0,Y 544.657,Z 630.315,A -85,B 0,C 180,E1 -3686.3,E2 -3686.3} C_VEL
LIN {X 0,Y 544.569,Z 633.001,A -85,B 0,C 180,E1 -3687.78,E2 -3687.78} C_VEL
LIN {X 0,Y 544.539,Z 634.333,A -85,B 0,C 180,E1 -3689.26,E2 -3689.26} C_VEL
LIN {X 0,Y 544.539,Z 634.334,A -85,B 0,C 180,E1 -3690.739,E2 -3690.739} C_VEL
LIN {X 0,Y 544.569,Z 633.005,A -85,B 0,C 180,E1 -3692.218,E2 -3692.218} C_VEL
LIN {X 0,Y 544.657,Z 630.322,A -85,B 0,C 180,E1 -3693.698,E2 -3693.698} C_VEL
LIN {X 0,Y 544.646,Z 626.204,A -85,B 0,C 180,E1 -3695.182,E2 -3695.182} C_VEL
LIN {X 0,Y 544.737,Z 620.939,A -85,B 0,C 180,E1 -3696.573,E2 -3696.573} C_VEL
LIN {X 0,Y 544.833,Z 614.131,A -85,B 0,C 180,E1 -3697.97,E2 -3697.97} C_VEL
LIN {X 0,Y 544.999,Z 606.179,A -85,B 0,C 180,E1 -3699.275,E2 -3699.275} C_VEL
LIN {X 0,Y 545.175,Z 597.858,A -85,B 0,C 180,E1 -3700.397,E2 -3700.397} C_VEL
LIN {X 0,Y 545.363,Z 588.035,A -85,B 0,C 180,E1 -3701.5,E2 -3701.5} C_VEL
LIN {X 0,Y 545.661,Z 576.657,A -85,B 0,C 180,E1 -3702.552,E2 -3702.552} C_VEL
LIN {X 0,Y 545.919,Z 564.112,A -85,B 0,C 180,E1 -3703.493,E2 -3703.493} C_VEL
LIN {X 0,Y 546.258,Z 551.652,A -85,B 0,C 180,E1 -3704.243,E2 -3704.243} C_VEL
LIN {X 0,Y 546.518,Z 537.712,A -85,B 0,C 180,E1 -3704.903,E2 -3704.903} C_VEL
LIN {X 0,Y 546.717,Z 523.724,A -85,B 0,C 180,E1 -3705.395,E2 -3705.395} C_VEL
LIN {X 0,Y 546.91,Z 509.879,A -85,B 0,C 180,E1 -3705.727,E2 -3705.727} C_VEL
LIN {X 0,Y 547.416,Z 380.087,A -85,B 0,C 180,E1 -3707.472,E2 -3707.472} C_VEL
LIN {X 0,Y 545.82,Z 371.025,A -85,B 0,C 180,E1 -3707.668,E2 -3707.668} C_VEL
LIN {X 0,Y 546.252,Z 349.438,A -85,B 0,C 180,E1 -3710.523,E2 -3710.523} C_VEL
LIN {X 0,Y 546.695,Z 324.967,A -85,B 0,C 180,E1 -3713.814,E2 -3713.814} C_VEL
LIN {X 0,Y 546.637,Z 318.568,A -85,B 0,C 180,E1 -3714.698,E2 -3714.698} C_VEL
LIN {X 0,Y 545.113,Z 311.21,A -85,B 0,C 180,E1 -3715.794,E2 -3715.794} C_VEL
LIN {X 0,Y 545.088,Z 311.214,A -85,B 0,C 180,E1 -3718.747,E2 -3718.747} C_VEL
LIN {X 0,Y 545.057,Z 311.212,A -85,B 0,C 180,E1 -3721.678,E2 -3721.678} C_VEL
LIN {X 0,Y 545.079,Z 311.212,A -85,B 0,C 180,E1 -3724.562,E2 -3724.562} C_VEL
LIN {X 0,Y 545.037,Z 311.216,A -85,B 0,C 180,E1 -3727.303,E2 -3727.303} C_VEL
LIN {X 0,Y 545.071,Z 311.211,A -85,B 0,C 180,E1 -3730.141,E2 -3730.141} C_VEL
LIN {X 0,Y 545.074,Z 311.213,A -85,B 0,C 180,E1 -3733.106,E2 -3733.106} C_VEL
LIN {X 0,Y 545.06,Z 311.211,A -85,B 0,C 180,E1 -3736.224,E2 -3736.224} C_VEL
LIN {X 0,Y 545.093,Z 311.209,A -85,B 0,C 180,E1 -3738.886,E2 -3738.886} C_VEL
LIN {X 0,Y 545.048,Z 311.211,A -85,B 0,C 180,E1 -3741.762,E2 -3741.762} C_VEL
LIN {X 0,Y 545.052,Z 311.219,A -85,B 0,C 180,E1 -3744.532,E2 -3744.532} C_VEL
LIN {X 0,Y 545.075,Z 311.207,A -85,B 0,C 180,E1 -3747.212,E2 -3747.212} C_VEL
LIN {X 0,Y 545.096,Z 311.207,A -85,B 0,C 180,E1 -3749.812,E2 -3749.812} C_VEL
LIN {X 0,Y 545.095,Z 311.207,A -85,B 0,C 180,E1 -3752.824,E2 -3752.824} C_VEL
LIN {X 0,Y 545.041,Z 311.214,A -85,B 0,C 180,E1 -3755.63,E2 -3755.63} C_VEL
LIN {X 0,Y 545.058,Z 311.212,A -85,B 0,C 180,E1 -3758.836,E2 -3758.836} C_VEL
LIN {X 0,Y 545.07,Z 311.207,A -85,B 0,C 180,E1 -3761.195,E2 -3761.195} C_VEL
LIN {X 0,Y 545.062,Z 311.212,A -85,B 0,C 180,E1 -3763.521,E2 -3763.521} C_VEL
LIN {X 0,Y 545.085,Z 311.211,A -85,B 0,C 180,E1 -3765.819,E2 -3765.819} C_VEL
LIN {X 0,Y 545.108,Z 311.202,A -85,B 0,C 180,E1 -3768.849,E2 -3768.849} C_VEL
LIN {X 0,Y 545.115,Z 311.212,A -85,B 0,C 180,E1 -3771.847,E2 -3771.847} C_VEL
LIN {X 0,Y 545.187,Z 311.194,A -85,B 0,C 180,E1 -3774.823,E2 -3774.823} C_VEL
LIN {X 0,Y 545.178,Z 311.202,A -85,B 0,C 180,E1 -3777.783,E2 -3777.783} C_VEL
LIN {X 0,Y 545.177,Z 311.199,A -85,B 0,C 180,E1 -3780,E2 -3780} C_VEL
LIN {X 0,Y 545.147,Z 311.2,A -85,B 0,C 180,E1 -3782.956,E2 -3782.956} C_VEL
LIN {X 0,Y 545.11,Z 311.208,A -85,B 0,C 180,E1 -3785.92,E2 -3785.92} C_VEL
LIN {X 0,Y 545.057,Z 311.211,A -85,B 0,C 180,E1 -3788.901,E2 -3788.901} C_VEL
LIN {X 0,Y 545.079,Z 311.209,A -85,B 0,C 180,E1 -3791.905,E2 -3791.905} C_VEL
LIN {X 0,Y 545.064,Z 311.213,A -85,B 0,C 180,E1 -3794.944,E2 -3794.944} C_VEL
LIN {X 0,Y 545.041,Z 311.213,A -85,B 0,C 180,E1 -3798.027,E2 -3798.027} C_VEL
LIN {X 0,Y 545.077,Z 311.208,A -85,B 0,C 180,E1 -3800.372,E2 -3800.372} C_VEL
LIN {X 0,Y 545.059,Z 311.215,A -85,B 0,C 180,E1 -3803.56,E2 -3803.56} C_VEL
LIN {X 0,Y 545.076,Z 311.213,A -85,B 0,C 180,E1 -3806.825,E2 -3806.825} C_VEL
LIN {X 0,Y 545.017,Z 311.222,A -85,B 0,C 180,E1 -3809.341,E2 -3809.341} C_VEL
LIN {X 0,Y 545.044,Z 311.213,A -85,B 0,C 180,E1 -3811.915,E2 -3811.915} C_VEL
LIN {X 0,Y 545.048,Z 311.216,A -85,B 0,C 180,E1 -3814.565,E2 -3814.565} C_VEL
LIN {X 0,Y 545.056,Z 311.217,A -85,B 0,C 180,E1 -3816.961,E2 -3816.961} C_VEL
LIN {X 0,Y 544.346,Z 311.304,A -85,B 0,C 180,E1 -3817.578,E2 -3817.578} C_VEL
LIN {X 0,Y 541.48,Z 311.662,A -85,B 0,C 180,E1 -3818.579,E2 -3818.579} C_VEL
LIN {X 0,Y 539.093,Z 311.956,A -85,B 0,C 180,E1 -3819.385,E2 -3819.385} C_VEL
LIN {X 0,Y 538.082,Z 312.079,A -85,B 0,C 180,E1 -3820.007,E2 -3820.007} C_VEL
LIN {X 0,Y 538.006,Z 312.09,A -85,B 0,C 180,E1 -3820.217,E2 -3820.217} C_VEL
LIN {X 0,Y 538.017,Z 312.095,A -85,B 0,C 180,E1 -3822.988,E2 -3822.988} C_VEL
LIN {X 0,Y 537.994,Z 312.093,A -85,B 0,C 180,E1 -3826.184,E2 -3826.184} C_VEL
LIN {X 0,Y 538.04,Z 312.09,A -85,B 0,C 180,E1 -3829.253,E2 -3829.253} C_VEL
LIN {X 0,Y 538.093,Z 312.275,A -85,B 0,C 180,E1 -3830.475,E2 -3830.475} C_VEL
LIN {X 0,Y 538.985,Z 317.768,A -85,B 0,C 180,E1 -3831.477,E2 -3831.477} C_VEL
LIN {X 0,Y 538.74,Z 331.455,A -85,B 0,C 180,E1 -3833.824,E2 -3833.824} C_VEL
LIN {X 0,Y 538.692,Z 333.575,A -85,B 0,C 180,E1 -3834.179,E2 -3834.179} C_VEL
LIN {X 0,Y 540.66,Z 343.215,A -85,B 0,C 180,E1 -3834.38,E2 -3834.38} C_VEL
LIN {X 0,Y 540.095,Z 470.175,A -85,B 0,C 180,E1 -3836.113,E2 -3836.113} C_VEL
LIN {X 0,Y 539.899,Z 484.653,A -85,B 0,C 180,E1 -3836.47,E2 -3836.47} C_VEL
LIN {X 0,Y 539.665,Z 498.145,A -85,B 0,C 180,E1 -3836.954,E2 -3836.954} C_VEL
LIN {X 0,Y 539.338,Z 511.604,A -85,B 0,C 180,E1 -3837.597,E2 -3837.597} C_VEL
LIN {X 0,Y 539.012,Z 524.182,A -85,B 0,C 180,E1 -3838.365,E2 -3838.365} C_VEL
LIN {X 0,Y 538.729,Z 535.298,A -85,B 0,C 180,E1 -3839.201,E2 -3839.201} C_VEL
LIN {X 0,Y 538.464,Z 545.835,A -85,B 0,C 180,E1 -3840.159,E2 -3840.159} C_VEL
LIN {X 0,Y 538.196,Z 556.413,A -85,B 0,C 180,E1 -3841.322,E2 -3841.322} C_VEL
LIN {X 0,Y 537.939,Z 565.547,A -85,B 0,C 180,E1 -3842.549,E2 -3842.549} C_VEL
LIN {X 0,Y 537.769,Z 573.381,A -85,B 0,C 180,E1 -3843.829,E2 -3843.829} C_VEL
LIN {X 0,Y 537.656,Z 578.621,A -85,B 0,C 180,E1 -3844.861,E2 -3844.861} C_VEL
LIN {X 0,Y 537.603,Z 584.236,A -85,B 0,C 180,E1 -3846.219,E2 -3846.219} C_VEL
LIN {X 0,Y 537.525,Z 588.934,A -85,B 0,C 180,E1 -3847.719,E2 -3847.719} C_VEL
LIN {X 0,Y 537.516,Z 590.828,A -85,B 0,C 180,E1 -3848.526,E2 -3848.526} C_VEL
LIN {X 0,Y 537.457,Z 593.388,A -85,B 0,C 180,E1 -3850.125,E2 -3850.125} C_VEL
LIN {X 0,Y 537.441,Z 594.435,A -85,B 0,C 180,E1 -3851.71,E2 -3851.71} C_VEL
LIN {X 0,Y 537.452,Z 594.025,A -85,B 0,C 180,E1 -3853.282,E2 -3853.282} C_VEL
LIN {X 0,Y 537.446,Z 592.184,A -85,B 0,C 180,E1 -3854.84,E2 -3854.84} C_VEL
LIN {X 0,Y 537.538,Z 588.881,A -85,B 0,C 180,E1 -3856.389,E2 -3856.389} C_VEL
LIN {X 0,Y 537.607,Z 584.025,A -85,B 0,C 180,E1 -3857.927,E2 -3857.927} C_VEL
LIN {X 0,Y 537.686,Z 579.346,A -85,B 0,C 180,E1 -3859.076,E2 -3859.076} C_VEL
LIN {X 0,Y 537.793,Z 572.562,A -85,B 0,C 180,E1 -3860.409,E2 -3860.409} C_VEL
LIN {X 0,Y 537.963,Z 564.171,A -85,B 0,C 180,E1 -3861.738,E2 -3861.738} C_VEL
LIN {X 0,Y 538.256,Z 554.419,A -85,B 0,C 180,E1 -3863.001,E2 -3863.001} C_VEL
LIN {X 0,Y 538.473,Z 545.047,A -85,B 0,C 180,E1 -3864.007,E2 -3864.007} C_VEL
LIN {X 0,Y 538.762,Z 533.397,A -85,B 0,C 180,E1 -3865.043,E2 -3865.043} C_VEL
LIN {X 0,Y 539.06,Z 521.736,A -85,B 0,C 180,E1 -3865.889,E2 -3865.889} C_VEL
LIN {X 0,Y 539.425,Z 508.872,A -85,B 0,C 180,E1 -3866.64,E2 -3866.64} C_VEL
LIN {X 0,Y 539.73,Z 495.432,A -85,B 0,C 180,E1 -3867.249,E2 -3867.249} C_VEL
LIN {X 0,Y 539.951,Z 481.336,A -85,B 0,C 180,E1 -3867.716,E2 -3867.716} C_VEL
LIN {X 0,Y 540.133,Z 467.606,A -85,B 0,C 180,E1 -3868.02,E2 -3868.02} C_VEL
LIN {X 0,Y 540.646,Z 343.215,A -85,B 0,C 180,E1 -3869.71,E2 -3869.71} C_VEL
LIN {X 0,Y 538.712,Z 333.432,A -85,B 0,C 180,E1 -3869.931,E2 -3869.931} C_VEL
LIN {X 0,Y 539.061,Z 317.66,A -85,B 0,C 180,E1 -3872.616,E2 -3872.616} C_VEL
LIN {X 0,Y 538,Z 312.098,A -85,B 0,C 180,E1 -3873.652,E2 -3873.652} C_VEL
LIN {X 0,Y 538.086,Z 312.083,A -85,B 0,C 180,E1 -3875.998,E2 -3875.998} C_VEL
LIN {X 0,Y 538.055,Z 312.085,A -85,B 0,C 180,E1 -3878.261,E2 -3878.261} C_VEL
LIN {X 0,Y 538.081,Z 312.084,A -85,B 0,C 180,E1 -3881.597,E2 -3881.597} C_VEL
LIN {X 0,Y 538.041,Z 312.087,A -85,B 0,C 180,E1 -3884.851,E2 -3884.851} C_VEL
LIN {X 0,Y 538.035,Z 312.089,A -85,B 0,C 180,E1 -3887.533,E2 -3887.533} C_VEL
LIN {X 0,Y 538.032,Z 312.087,A -85,B 0,C 180,E1 -3890.652,E2 -3890.652} C_VEL
LIN {X 0,Y 538.005,Z 312.089,A -85,B 0,C 180,E1 -3893.878,E2 -3893.878} C_VEL
LIN {X 0,Y 537.98,Z 312.092,A -85,B 0,C 180,E1 -3896.37,E2 -3896.37} C_VEL
LIN {X 0,Y 537.99,Z 312.098,A -85,B 0,C 180,E1 -3898.926,E2 -3898.926} C_VEL
LIN {X 0,Y 537.993,Z 312.09,A -85,B 0,C 180,E1 -3901.885,E2 -3901.885} C_VEL
LIN {X 0,Y 537.99,Z 312.095,A -85,B 0,C 180,E1 -3904.615,E2 -3904.615} C_VEL
LIN {X 0,Y 537.965,Z 312.093,A -85,B 0,C 180,E1 -3907.88,E2 -3907.88} C_VEL
LIN {X 0,Y 537.995,Z 312.099,A -85,B 0,C 180,E1 -3910.781,E2 -3910.781} C_VEL
LIN {X 0,Y 537.991,Z 312.091,A -85,B 0,C 180,E1 -3914.071,E2 -3914.071} C_VEL
LIN {X 0,Y 537.952,Z 312.1,A -85,B 0,C 180,E1 -3917.021,E2 -3917.021} C_VEL
LIN {X 0,Y 537.987,Z 312.092,A -85,B 0,C 180,E1 -3919.261,E2 -3919.261} C_VEL
LIN {X 0,Y 537.963,Z 312.096,A -85,B 0,C 180,E1 -3922.12,E2 -3922.12} C_VEL
LIN {X 0,Y 537.994,Z 312.09,A -85,B 0,C 180,E1 -3925.386,E2 -3925.386} C_VEL
LIN {X 0,Y 537.999,Z 312.092,A -85,B 0,C 180,E1 -3928.115,E2 -3928.115} C_VEL
LIN {X 0,Y 537.984,Z 312.092,A -85,B 0,C 180,E1 -3931.096,E2 -3931.096} C_VEL
LIN {X 0,Y 537.984,Z 312.091,A -85,B 0,C 180,E1 -3933.631,E2 -3933.631} C_VEL
LIN {X 0,Y 537.984,Z 312.096,A -85,B 0,C 180,E1 -3936.128,E2 -3936.128} C_VEL
LIN {X 0,Y 538.02,Z 312.086,A -85,B 0,C 180,E1 -3939.348,E2 -3939.348} C_VEL
LIN {X 0,Y 538.014,Z 312.094,A -85,B 0,C 180,E1 -3942.476,E2 -3942.476} C_VEL
LIN {X 0,Y 538.044,Z 312.085,A -85,B 0,C 180,E1 -3945.63,E2 -3945.63} C_VEL
LIN {X 0,Y 538.078,Z 312.082,A -85,B 0,C 180,E1 -3948.702,E2 -3948.702} C_VEL
LIN {X 0,Y 538.059,Z 312.085,A -85,B 0,C 180,E1 -3951.739,E2 -3951.739} C_VEL
LIN {X 0,Y 538.152,Z 312.071,A -85,B 0,C 180,E1 -3954.755,E2 -3954.755} C_VEL
LIN {X 0,Y 538.167,Z 312.073,A -85,B 0,C 180,E1 -3957.755,E2 -3957.755} C_VEL
LIN {X 0,Y 538.181,Z 312.067,A -85,B 0,C 180,E1 -3960.748,E2 -3960.748} C_VEL
LIN {X 0,Y 538.127,Z 312.073,A -85,B 0,C 180,E1 -3962.995,E2 -3962.995} C_VEL
LIN {X 0,Y 538.115,Z 312.083,A -85,B 0,C 180,E1 -3965.998,E2 -3965.998} C_VEL
LIN {X 0,Y 538.062,Z 312.082,A -85,B 0,C 180,E1 -3969.018,E2 -3969.018} C_VEL
LIN {X 0,Y 538.067,Z 312.086,A -85,B 0,C 180,E1 -3972.063,E2 -3972.063} C_VEL
LIN {X 0,Y 538.048,Z 312.085,A -85,B 0,C 180,E1 -3975.144,E2 -3975.144} C_VEL
LIN {X 0,Y 538.031,Z 312.087,A -85,B 0,C 180,E1 -3978.27,E2 -3978.27} C_VEL
LIN {X 0,Y 538.042,Z 312.084,A -85,B 0,C 180,E1 -3980.651,E2 -3980.651} C_VEL
LIN {X 0,Y 538.005,Z 312.093,A -85,B 0,C 180,E1 -3983.889,E2 -3983.889} C_VEL
LIN {X 0,Y 538.043,Z 312.084,A -85,B 0,C 180,E1 -3986.367,E2 -3986.367} C_VEL
LIN {X 0,Y 538.034,Z 312.087,A -85,B 0,C 180,E1 -3988.933,E2 -3988.933} C_VEL
LIN {X 0,Y 538.014,Z 312.09,A -85,B 0,C 180,E1 -3991.887,E2 -3991.887} C_VEL
LIN {X 0,Y 538.014,Z 312.088,A -85,B 0,C 180,E1 -3994.617,E2 -3994.617} C_VEL
LIN {X 0,Y 538.003,Z 312.095,A -85,B 0,C 180,E1 -3997.169,E2 -3997.169} C_VEL
LIN {X 0,Y 538.025,Z 312.089,A -85,B 0,C 180,E1 -3999.797,E2 -3999.797} C_VEL
LIN {X 0,Y 538.023,Z 312.089,A -85,B 0,C 180,E1 -4002.786,E2 -4002.786} C_VEL
LIN {X 0,Y 538.023,Z 312.087,A -85,B 0,C 180,E1 -4005.927,E2 -4005.927} C_VEL
LIN {X 0,Y 538.034,Z 312.085,A -85,B 0,C 180,E1 -4008.227,E2 -4008.227} C_VEL
LIN {X 0,Y 538.019,Z 312.096,A -85,B 0,C 180,E1 -4011.17,E2 -4011.17} C_VEL
LIN {X 0,Y 537.998,Z 312.089,A -85,B 0,C 180,E1 -4014.088,E2 -4014.088} C_VEL
LIN {X 0,Y 538.034,Z 312.089,A -85,B 0,C 180,E1 -4016.727,E2 -4016.727} C_VEL
LIN {X 0,Y 538.018,Z 312.092,A -85,B 0,C 180,E1 -4019.558,E2 -4019.558} C_VEL
LIN {X 0,Y 538.044,Z 312.089,A -85,B 0,C 180,E1 -4021.95,E2 -4021.95} C_VEL
LIN {X 0,Y 538.096,Z 312.167,A -85,B 0,C 180,E1 -4024.001,E2 -4024.001} C_VEL
LIN {X 0,Y 539.937,Z 321.38,A -85,B 0,C 180,E1 -4025.384,E2 -4025.384} C_VEL
LIN {X 0,Y 539.461,Z 343.38,A -85,B 0,C 180,E1 -4028.405,E2 -4028.405} C_VEL
LIN {X 0,Y 538.985,Z 365.352,A -85,B 0,C 180,E1 -4031.369,E2 -4031.369} C_VEL
LIN {X 0,Y 538.86,Z 371.06,A -85,B 0,C 180,E1 -4032.122,E2 -4032.122} C_VEL
LIN {X 0,Y 540.63,Z 381.199,A -85,B 0,C 180,E1 -4032.32,E2 -4032.32} C_VEL
LIN {X 0,Y 540.123,Z 509.494,A -85,B 0,C 180,E1 -4034.069,E2 -4034.069} C_VEL
LIN {X 0,Y 539.849,Z 524.005,A -85,B 0,C 180,E1 -4034.423,E2 -4034.423} C_VEL
LIN {X 0,Y 539.606,Z 538.566,A -85,B 0,C 180,E1 -4034.949,E2 -4034.949} C_VEL
LIN {X 0,Y 539.33,Z 551.429,A -85,B 0,C 180,E1 -4035.568,E2 -4035.568} C_VEL
LIN {X 0,Y 538.988,Z 563.952,A -85,B 0,C 180,E1 -4036.329,E2 -4036.329} C_VEL
LIN {X 0,Y 538.686,Z 576.58,A -85,B 0,C 180,E1 -4037.281,E2 -4037.281} C_VEL
LIN {X 0,Y 538.435,Z 586.814,A -85,B 0,C 180,E1 -4038.223,E2 -4038.223} C_VEL
LIN {X 0,Y 538.205,Z 596.328,A -85,B 0,C 180,E1 -4039.275,E2 -4039.275} C_VEL
LIN {X 0,Y 537.968,Z 604.905,A -85,B 0,C 180,E1 -4040.411,E2 -4040.411} C_VEL
LIN {X 0,Y 537.805,Z 613.115,A -85,B 0,C 180,E1 -4041.735,E2 -4041.735} C_VEL
LIN {X 0,Y 537.662,Z 618.86,A -85,B 0,C 180,E1 -4042.866,E2 -4042.866} C_VEL
LIN {X 0,Y 537.656,Z 624.958,A -85,B 0,C 180,E1 -4044.373,E2 -4044.373} C_VEL
LIN {X 0,Y 537.55,Z 628.442,A -85,B 0,C 180,E1 -4045.5,E2 -4045.5} C_VEL
LIN {X 0,Y 537.547,Z 631.831,A -85,B 0,C 180,E1 -4047.002,E2 -4047.002} C_VEL
LIN {X 0,Y 537.447,Z 633.834,A -85,B 0,C 180,E1 -4048.501,E2 -4048.501} C_VEL
LIN {X 0,Y 537.44,Z 634.5,A -85,B 0,C 180,E1 -4049.999,E2 -4049.999} C_VEL
LIN {X 0,Y 537.447,Z 633.837,A -85,B 0,C 180,E1 -4051.498,E2 -4051.498} C_VEL
LIN {X 0,Y 537.547,Z 631.837,A -85,B 0,C 180,E1 -4052.997,E2 -4052.997} C_VEL
LIN {X 0,Y 537.55,Z 628.449,A -85,B 0,C 180,E1 -4054.498,E2 -4054.498} C_VEL
LIN {X 0,Y 537.65,Z 623.57,A -85,B 0,C 180,E1 -4056.002,E2 -4056.002} C_VEL
LIN {X 0,Y 537.704,Z 617.057,A -85,B 0,C 180,E1 -4057.51,E2 -4057.51} C_VEL
LIN {X 0,Y 537.858,Z 609.808,A -85,B 0,C 180,E1 -4058.831,E2 -4058.831} C_VEL
LIN {X 0,Y 538.063,Z 600.827,A -85,B 0,C 180,E1 -4060.155,E2 -4060.155} C_VEL
LIN {X 0,Y 538.341,Z 591.399,A -85,B 0,C 180,E1 -4061.292,E2 -4061.292} C_VEL
LIN {X 0,Y 538.546,Z 580.92,A -85,B 0,C 180,E1 -4062.338,E2 -4062.338} C_VEL
LIN {X 0,Y 538.85,Z 569.325,A -85,B 0,C 180,E1 -4063.289,E2 -4063.289} C_VEL
LIN {X 0,Y 539.184,Z 556.467,A -85,B 0,C 180,E1 -4064.145,E2 -4064.145} C_VEL
LIN {X 0,Y 539.527,Z 542.917,A -85,B 0,C 180,E1 -4064.859,E2 -4064.859} C_VEL
LIN {X 0,Y 539.806,Z 529.821,A -85,B 0,C 180,E1 -4065.387,E2 -4065.387} C_VEL
LIN {X 0,Y 540.025,Z 515.908,A -85,B 0,C 180,E1 -4065.795,E2 -4065.795} C_VEL
LIN {X 0,Y 540.135,Z 500.437,A -85,B 0,C 180,E1 -4066.075,E2 -4066.075} C_VEL
LIN {X 0,Y 540.603,Z 380.74,A -85,B 0,C 180,E1 -4067.687,E2 -4067.687} C_VEL
LIN {X 0,Y 538.861,Z 370.773,A -85,B 0,C 180,E1 -4067.899,E2 -4067.899} C_VEL
LIN {X 0,Y 539.379,Z 347.708,A -85,B 0,C 180,E1 -4070.996,E2 -4070.996} C_VEL
LIN {X 0,Y 539.941,Z 322.713,A -85,B 0,C 180,E1 -4074.412,E2 -4074.412} C_VEL
LIN {X 0,Y 539.396,Z 318.312,A -85,B 0,C 180,E1 -4075.052,E2 -4075.052} C_VEL
LIN {X 0,Y 538.069,Z 312.087,A -85,B 0,C 180,E1 -4075.999,E2 -4075.999} C_VEL
LIN {X 0,Y 538.029,Z 312.094,A -85,B 0,C 180,E1 -4078.933,E2 -4078.933} C_VEL
LIN {X 0,Y 538.012,Z 312.089,A -85,B 0,C 180,E1 -4081.887,E2 -4081.887} C_VEL
LIN {X 0,Y 538.029,Z 312.091,A -85,B 0,C 180,E1 -4084.62,E2 -4084.62} C_VEL
LIN {X 0,Y 538.005,Z 312.094,A -85,B 0,C 180,E1 -4087.17,E2 -4087.17} C_VEL
LIN {X 0,Y 538.026,Z 312.087,A -85,B 0,C 180,E1 -4089.795,E2 -4089.795} C_VEL
LIN {X 0,Y 538.033,Z 312.084,A -85,B 0,C 180,E1 -4091.879,E2 -4091.879} C_VEL
LIN {X 0,Y 538.028,Z 312.086,A -85,B 0,C 180,E1 -4095.14,E2 -4095.14} C_VEL
LIN {X 0,Y 538.036,Z 312.089,A -85,B 0,C 180,E1 -4098.227,E2 -4098.227} C_VEL
LIN {X 0,Y 538.01,Z 312.088,A -85,B 0,C 180,E1 -4101.169,E2 -4101.169} C_VEL
LIN {X 0,Y 538.021,Z 312.091,A -85,B 0,C 180,E1 -4104.083,E2 -4104.083} C_VEL
LIN {X 0,Y 538.024,Z 312.09,A -85,B 0,C 180,E1 -4106.727,E2 -4106.727} C_VEL
LIN {X 0,Y 538.032,Z 312.086,A -85,B 0,C 180,E1 -4109.553,E2 -4109.553} C_VEL
LIN {X 0,Y 538.042,Z 312.088,A -85,B 0,C 180,E1 -4111.95,E2 -4111.95} C_VEL
LIN {X 0,Y 538.069,Z 312.087,A -85,B 0,C 180,E1 -4114.467,E2 -4114.467} C_VEL
LIN {X 0,Y 537.985,Z 312.092,A -85,B 0,C 180,E1 -4117.738,E2 -4117.738} C_VEL
LIN {X 0,Y 538.072,Z 312.088,A -85,B 0,C 180,E1 -4120.147,E2 -4120.147} C_VEL
LIN {X 0,Y 538.014,Z 312.088,A -85,B 0,C 180,E1 -4123.298,E2 -4123.298} C_VEL
LIN {X 0,Y 538.054,Z 312.084,A -85,B 0,C 180,E1 -4125.63,E2 -4125.63} C_VEL
LIN {X 0,Y 538.068,Z 312.079,A -85,B 0,C 180,E1 -4128.701,E2 -4128.701} C_VEL
LIN {X 0,Y 538.072,Z 312.088,A -85,B 0,C 180,E1 -4131.739,E2 -4131.739} C_VEL
LIN {X 0,Y 538.104,Z 312.084,A -85,B 0,C 180,E1 -4134.002,E2 -4134.002} C_VEL
LIN {X 0,Y 538.113,Z 312.074,A -85,B 0,C 180,E1 -4137.005,E2 -4137.005} C_VEL
LIN {X 0,Y 538.146,Z 312.075,A -85,B 0,C 180,E1 -4140,E2 -4140} C_VEL
LIN {X 0,Y 538.115,Z 312.076,A -85,B 0,C 180,E1 -4142.994,E2 -4142.994} C_VEL
LIN {X 0,Y 538.062,Z 312.085,A -85,B 0,C 180,E1 -4145.998,E2 -4145.998} C_VEL
LIN {X 0,Y 538.015,Z 312.089,A -85,B 0,C 180,E1 -4149.018,E2 -4149.018} C_VEL
LIN {X 0,Y 538.038,Z 312.085,A -85,B 0,C 180,E1 -4152.063,E2 -4152.063} C_VEL
LIN {X 0,Y 538.025,Z 312.092,A -85,B 0,C 180,E1 -4155.144,E2 -4155.144} C_VEL
LIN {X 0,Y 537.994,Z 312.09,A -85,B 0,C 180,E1 -4158.271,E2 -4158.271} C_VEL
LIN {X 0,Y 538.021,Z 312.088,A -85,B 0,C 180,E1 -4160.652,E2 -4160.652} C_VEL
LIN {X 0,Y 537.995,Z 312.091,A -85,B 0,C 180,E1 -4163.878,E2 -4163.878} C_VEL
LIN {X 0,Y 538.021,Z 312.088,A -85,B 0,C 180,E1 -4166.367,E2 -4166.367} C_VEL
LIN {X 0,Y 537.981,Z 312.095,A -85,B 0,C 180,E1 -4168.926,E2 -4168.926} C_VEL
LIN {X 0,Y 537.999,Z 312.091,A -85,B 0,C 180,E1 -4171.887,E2 -4171.887} C_VEL
LIN {X 0,Y 537.998,Z 312.095,A -85,B 0,C 180,E1 -4174.617,E2 -4174.617} C_VEL
LIN {X 0,Y 537.994,Z 312.097,A -85,B 0,C 180,E1 -4177.17,E2 -4177.17} C_VEL
LIN {X 0,Y 538.006,Z 312.09,A -85,B 0,C 180,E1 -4180.217,E2 -4180.217} C_VEL
LIN {X 0,Y 537.355,Z 312.179,A -85,B 0,C 180,E1 -4180.842,E2 -4180.842} C_VEL
LIN {X 0,Y 534.507,Z 312.532,A -85,B 0,C 180,E1 -4181.857,E2 -4181.857} C_VEL
LIN {X 0,Y 532.084,Z 312.832,A -85,B 0,C 180,E1 -4182.674,E2 -4182.674} C_VEL
LIN {X 0,Y 531.034,Z 312.961,A -85,B 0,C 180,E1 -4183.305,E2 -4183.305} C_VEL
LIN {X 0,Y 530.944,Z 312.97,A -85,B 0,C 180,E1 -4183.519,E2 -4183.519} C_VEL
LIN {X 0,Y 530.946,Z 312.975,A -85,B 0,C 180,E1 -4186.505,E2 -4186.505} C_VEL
LIN {X 0,Y 530.979,Z 312.969,A -85,B 0,C 180,E1 -4189.568,E2 -4189.568} C_VEL
LIN {X 0,Y 531.025,Z 312.997,A -85,B 0,C 180,E1 -4190.262,E2 -4190.262} C_VEL
LIN {X 0,Y 532.064,Z 319.271,A -85,B 0,C 180,E1 -4191.419,E2 -4191.419} C_VEL
LIN {X 0,Y 531.822,Z 332.553,A -85,B 0,C 180,E1 -4193.717,E2 -4193.717} C_VEL
LIN {X 0,Y 531.769,Z 333.765,A -85,B 0,C 180,E1 -4193.923,E2 -4193.923} C_VEL
LIN {X 0,Y 533.941,Z 344.671,A -85,B 0,C 180,E1 -4194.167,E2 -4194.167} C_VEL
LIN {X 0,Y 533.299,Z 469.996,A -85,B 0,C 180,E1 -4195.897,E2 -4195.897} C_VEL
LIN {X 0,Y 533.077,Z 484.735,A -85,B 0,C 180,E1 -4196.261,E2 -4196.261} C_VEL
LIN {X 0,Y 532.835,Z 498.426,A -85,B 0,C 180,E1 -4196.757,E2 -4196.757} C_VEL
LIN {X 0,Y 532.455,Z 512.35,A -85,B 0,C 180,E1 -4197.434,E2 -4197.434} C_VEL
LIN {X 0,Y 532.092,Z 524.968,A -85,B 0,C 180,E1 -4198.22,E2 -4198.22} C_VEL
LIN {X 0,Y 531.777,Z 536.862,A -85,B 0,C 180,E1 -4199.139,E2 -4199.139} C_VEL
LIN {X 0,Y 531.486,Z 547.719,A -85,B 0,C 180,E1 -4200.165,E2 -4200.165} C_VEL
LIN {X 0,Y 531.177,Z 557.943,A -85,B 0,C 180,E1 -4201.34,E2 -4201.34} C_VEL
LIN {X 0,Y 530.87,Z 567.313,A -85,B 0,C 180,E1 -4202.657,E2 -4202.657} C_VEL
LIN {X 0,Y 530.703,Z 574.411,A -85,B 0,C 180,E1 -4203.876,E2 -4203.876} C_VEL
LIN {X 0,Y 530.55,Z 581.262,A -85,B 0,C 180,E1 -4205.339,E2 -4205.339} C_VEL
LIN {X 0,Y 530.511,Z 585.841,A -85,B 0,C 180,E1 -4206.583,E2 -4206.583} C_VEL
LIN {X 0,Y 530.44,Z 589.896,A -85,B 0,C 180,E1 -4208.041,E2 -4208.041} C_VEL
LIN {X 0,Y 530.368,Z 591.934,A -85,B 0,C 180,E1 -4209.037,E2 -4209.037} C_VEL
LIN {X 0,Y 530.372,Z 593.958,A -85,B 0,C 180,E1 -4210.655,E2 -4210.655} C_VEL
LIN {X 0,Y 530.367,Z 594.476,A -85,B 0,C 180,E1 -4212.256,E2 -4212.256} C_VEL
LIN {X 0,Y 530.332,Z 593.566,A -85,B 0,C 180,E1 -4213.842,E2 -4213.842} C_VEL
LIN {X 0,Y 530.403,Z 591.236,A -85,B 0,C 180,E1 -4215.419,E2 -4215.419} C_VEL
LIN {X 0,Y 530.467,Z 587.464,A -85,B 0,C 180,E1 -4216.985,E2 -4216.985} C_VEL
LIN {X 0,Y 530.518,Z 583.6,A -85,B 0,C 180,E1 -4218.152,E2 -4218.152} C_VEL
LIN {X 0,Y 530.597,Z 578.83,A -85,B 0,C 180,E1 -4219.314,E2 -4219.314} C_VEL
LIN {X 0,Y 530.76,Z 571.933,A -85,B 0,C 180,E1 -4220.666,E2 -4220.666} C_VEL
LIN {X 0,Y 530.977,Z 563.414,A -85,B 0,C 180,E1 -4222.012,E2 -4222.012} C_VEL
LIN {X 0,Y 531.259,Z 554.538,A -85,B 0,C 180,E1 -4223.163,E2 -4223.163} C_VEL
LIN {X 0,Y 531.541,Z 543.854,A -85,B 0,C 180,E1 -4224.31,E2 -4224.31} C_VEL
LIN {X 0,Y 531.834,Z 533.065,A -85,B 0,C 180,E1 -4225.263,E2 -4225.263} C_VEL
LIN {X 0,Y 532.219,Z 521.245,A -85,B 0,C 180,E1 -4226.12,E2 -4226.12} C_VEL
LIN {X 0,Y 532.615,Z 508.155,A -85,B 0,C 180,E1 -4226.881,E2 -4226.881} C_VEL
LIN {X 0,Y 532.899,Z 495.614,A -85,B 0,C 180,E1 -4227.45,E2 -4227.45} C_VEL
LIN {X 0,Y 533.134,Z 481.487,A -85,B 0,C 180,E1 -4227.923,E2 -4227.923} C_VEL
LIN {X 0,Y 533.322,Z 467.702,A -85,B 0,C 180,E1 -4228.231,E2 -4228.231} C_VEL
LIN {X 0,Y 533.907,Z 344.198,A -85,B 0,C 180,E1 -4229.93,E2 -4229.93} C_VEL
LIN {X 0,Y 531.791,Z 333.725,A -85,B 0,C 180,E1 -4230.166,E2 -4230.166} C_VEL
LIN {X 0,Y 532.149,Z 319.299,A -85,B 0,C 180,E1 -4232.65,E2 -4232.65} C_VEL
LIN {X 0,Y 530.952,Z 312.976,A -85,B 0,C 180,E1 -4233.843,E2 -4233.843} C_VEL
LIN {X 0,Y 531.046,Z 312.96,A -85,B 0,C 180,E1 -4236.078,E2 -4236.078} C_VEL
LIN {X 0,Y 531.006,Z 312.968,A -85,B 0,C 180,E1 -4239.139,E2 -4239.139} C_VEL
LIN {X 0,Y 531.024,Z 312.958,A -85,B 0,C 180,E1 -4242.226,E2 -4242.226} C_VEL
LIN {X 0,Y 530.988,Z 312.97,A -85,B 0,C 180,E1 -4245.351,E2 -4245.351} C_VEL
LIN {X 0,Y 530.97,Z 312.966,A -85,B 0,C 180,E1 -4248.522,E2 -4248.522} C_VEL
LIN {X 0,Y 530.994,Z 312.968,A -85,B 0,C 180,E1 -4250.939,E2 -4250.939} C_VEL
LIN {X 0,Y 530.947,Z 312.968,A -85,B 0,C 180,E1 -4254.227,E2 -4254.227} C_VEL
LIN {X 0,Y 530.944,Z 312.973,A -85,B 0,C 180,E1 -4256.747,E2 -4256.747} C_VEL
LIN {X 0,Y 530.953,Z 312.971,A -85,B 0,C 180,E1 -4259.325,E2 -4259.325} C_VEL
LIN {X 0,Y 530.949,Z 312.967,A -85,B 0,C 180,E1 -4262.098,E2 -4262.098} C_VEL
LIN {X 0,Y 530.952,Z 312.975,A -85,B 0,C 180,E1 -4264.849,E2 -4264.849} C_VEL
LIN {X 0,Y 530.923,Z 312.972,A -85,B 0,C 180,E1 -4267.512,E2 -4267.512} C_VEL
LIN {X 0,Y 530.942,Z 312.972,A -85,B 0,C 180,E1 -4270.437,E2 -4270.437} C_VEL
LIN {X 0,Y 530.917,Z 312.972,A -85,B 0,C 180,E1 -4273.5,E2 -4273.5} C_VEL
LIN {X 0,Y 530.958,Z 312.966,A -85,B 0,C 180,E1 -4275.625,E2 -4275.625} C_VEL
LIN {X 0,Y 530.925,Z 312.975,A -85,B 0,C 180,E1 -4278.984,E2 -4278.984} C_VEL
LIN {X 0,Y 530.92,Z 312.971,A -85,B 0,C 180,E1 -4281.527,E2 -4281.527} C_VEL
LIN {X 0,Y 530.927,Z 312.976,A -85,B 0,C 180,E1 -4284.378,E2 -4284.378} C_VEL
LIN {X 0,Y 530.964,Z 312.967,A -85,B 0,C 180,E1 -4287.134,E2 -4287.134} C_VEL
LIN {X 0,Y 530.93,Z 312.971,A -85,B 0,C 180,E1 -4289.801,E2 -4289.801} C_VEL
LIN {X 0,Y 530.955,Z 312.976,A -85,B 0,C 180,E1 -4292.48,E2 -4292.48} C_VEL
LIN {X 0,Y 530.948,Z 312.97,A -85,B 0,C 180,E1 -4294.94,E2 -4294.94} C_VEL
LIN {X 0,Y 530.952,Z 312.975,A -85,B 0,C 180,E1 -4298.246,E2 -4298.246} C_VEL
LIN {X 0,Y 530.97,Z 312.969,A -85,B 0,C 180,E1 -4300.677,E2 -4300.677} C_VEL
LIN {X 0,Y 530.93,Z 312.97,A -85,B 0,C 180,E1 -4303.069,E2 -4303.069} C_VEL
LIN {X 0,Y 531.003,Z 312.961,A -85,B 0,C 180,E1 -4305.436,E2 -4305.436} C_VEL
LIN {X 0,Y 531.036,Z 312.96,A -85,B 0,C 180,E1 -4308.55,E2 -4308.55} C_VEL
LIN {X 0,Y 531.035,Z 312.959,A -85,B 0,C 180,E1 -4311.629,E2 -4311.629} C_VEL
LIN {X 0,Y 531.111,Z 312.949,A -85,B 0,C 180,E1 -4314.685,E2 -4314.685} C_VEL
LIN {X 0,Y 531.139,Z 312.948,A -85,B 0,C 180,E1 -4317.725,E2 -4317.725} C_VEL
LIN {X 0,Y 531.152,Z 312.943,A -85,B 0,C 180,E1 -4320.758,E2 -4320.758} C_VEL
LIN {X 0,Y 531.093,Z 312.949,A -85,B 0,C 180,E1 -4323.034,E2 -4323.034} C_VEL
LIN {X 0,Y 531.07,Z 312.959,A -85,B 0,C 180,E1 -4326.077,E2 -4326.077} C_VEL
LIN {X 0,Y 531.054,Z 312.956,A -85,B 0,C 180,E1 -4328.371,E2 -4328.371} C_VEL
LIN {X 0,Y 531.053,Z 312.962,A -85,B 0,C 180,E1 -4331.671,E2 -4331.671} C_VEL
LIN {X 0,Y 531.035,Z 312.957,A -85,B 0,C 180,E1 -4334.956,E2 -4334.956} C_VEL
LIN {X 0,Y 531.02,Z 312.968,A -85,B 0,C 180,E1 -4337.722,E2 -4337.722} C_VEL
LIN {X 0,Y 531.003,Z 312.961,A -85,B 0,C 180,E1 -4340.938,E2 -4340.938} C_VEL
LIN {X 0,Y 530.968,Z 312.966,A -85,B 0,C 180,E1 -4344.225,E2 -4344.225} C_VEL
LIN {X 0,Y 531.001,Z 312.961,A -85,B 0,C 180,E1 -4346.744,E2 -4346.744} C_VEL
LIN {X 0,Y 530.985,Z 312.969,A -85,B 0,C 180,E1 -4349.323,E2 -4349.323} C_VEL
LIN {X 0,Y 530.969,Z 312.966,A -85,B 0,C 180,E1 -4352.1,E2 -4352.1} C_VEL
LIN {X 0,Y 530.972,Z 312.966,A -85,B 0,C 180,E1 -4354.851,E2 -4354.851} C_VEL
LIN {X 0,Y 530.967,Z 312.972,A -85,B 0,C 180,E1 -4357.508,E2 -4357.508} C_VEL
LIN {X 0,Y 530.984,Z 312.963,A -85,B 0,C 180,E1 -4360.433,E2 -4360.433} C_VEL
LIN {X 0,Y 530.968,Z 312.974,A -85,B 0,C 180,E1 -4363.281,E2 -4363.281} C_VEL
LIN {X 0,Y 530.985,Z 312.966,A -85,B 0,C 180,E1 -4365.621,E2 -4365.621} C_VEL
LIN {X 0,Y 530.997,Z 312.963,A -85,B 0,C 180,E1 -4368.564,E2 -4368.564} C_VEL
LIN {X 0,Y 530.963,Z 312.969,A -85,B 0,C 180,E1 -4371.529,E2 -4371.529} C_VEL
LIN {X 0,Y 530.959,Z 312.967,A -85,B 0,C 180,E1 -4374.38,E2 -4374.38} C_VEL
LIN {X 0,Y 530.971,Z 312.973,A -85,B 0,C 180,E1 -4377.133,E2 -4377.133} C_VEL
LIN {X 0,Y 530.965,Z 312.97,A -85,B 0,C 180,E1 -4379.802,E2 -4379.802} C_VEL
LIN {X 0,Y 531.017,Z 312.968,A -85,B 0,C 180,E1 -4382.467,E2 -4382.467} C_VEL
LIN {X 0,Y 531.049,Z 313.115,A -85,B 0,C 180,E1 -4383.799,E2 -4383.799} C_VEL
LIN {X 0,Y 533.065,Z 323.09,A -85,B 0,C 180,E1 -4385.319,E2 -4385.319} C_VEL
LIN {X 0,Y 532.521,Z 344.589,A -85,B 0,C 180,E1 -4388.313,E2 -4388.313} C_VEL
LIN {X 0,Y 531.986,Z 366.548,A -85,B 0,C 180,E1 -4391.315,E2 -4391.315} C_VEL
LIN {X 0,Y 531.903,Z 370.687,A -85,B 0,C 180,E1 -4391.876,E2 -4391.876} C_VEL
LIN {X 0,Y 533.86,Z 382.364,A -85,B 0,C 180,E1 -4392.108,E2 -4392.108} C_VEL
LIN {X 0,Y 533.289,Z 509.168,A -85,B 0,C 180,E1 -4393.859,E2 -4393.859} C_VEL
LIN {X 0,Y 533.033,Z 523.375,A -85,B 0,C 180,E1 -4394.208,E2 -4394.208} C_VEL
LIN {X 0,Y 532.772,Z 537.138,A -85,B 0,C 180,E1 -4394.702,E2 -4394.702} C_VEL
LIN {X 0,Y 532.457,Z 549.367,A -85,B 0,C 180,E1 -4395.28,E2 -4395.28} C_VEL
LIN {X 0,Y 532.111,Z 562.235,A -85,B 0,C 180,E1 -4396.051,E2 -4396.051} C_VEL
LIN {X 0,Y 531.775,Z 573.939,A -85,B 0,C 180,E1 -4396.919,E2 -4396.919} C_VEL
LIN {X 0,Y 531.454,Z 585.02,A -85,B 0,C 180,E1 -4397.916,E2 -4397.916} C_VEL
LIN {X 0,Y 531.217,Z 594.482,A -85,B 0,C 180,E1 -4398.94,E2 -4398.94} C_VEL
LIN {X 0,Y 530.926,Z 603.398,A -85,B 0,C 180,E1 -4400.09,E2 -4400.09} C_VEL
LIN {X 0,Y 530.757,Z 611.948,A -85,B 0,C 180,E1 -4401.432,E2 -4401.432} C_VEL
LIN {X 0,Y 530.587,Z 618.838,A -85,B 0,C 180,E1 -4402.77,E2 -4402.77} C_VEL
LIN {X 0,Y 530.551,Z 623.566,A -85,B 0,C 180,E1 -4403.916,E2 -4403.916} C_VEL
LIN {X 0,Y 530.449,Z 628.441,A -85,B 0,C 180,E1 -4405.44,E2 -4405.44} C_VEL
LIN {X 0,Y 530.452,Z 631.83,A -85,B 0,C 180,E1 -4406.961,E2 -4406.961} C_VEL
LIN {X 0,Y 530.357,Z 633.835,A -85,B 0,C 180,E1 -4408.481,E2 -4408.481} C_VEL
LIN {X 0,Y 530.341,Z 634.5,A -85,B 0,C 180,E1 -4409.999,E2 -4409.999} C_VEL
LIN {X 0,Y 530.357,Z 633.837,A -85,B 0,C 180,E1 -4411.518,E2 -4411.518} C_VEL
LIN {X 0,Y 530.452,Z 631.837,A -85,B 0,C 180,E1 -4413.037,E2 -4413.037} C_VEL
LIN {X 0,Y 530.449,Z 628.448,A -85,B 0,C 180,E1 -4414.559,E2 -4414.559} C_VEL
LIN {X 0,Y 530.546,Z 623.57,A -85,B 0,C 180,E1 -4416.083,E2 -4416.083} C_VEL
LIN {X 0,Y 530.585,Z 618.842,A -85,B 0,C 180,E1 -4417.228,E2 -4417.228} C_VEL
LIN {X 0,Y 530.755,Z 611.954,A -85,B 0,C 180,E1 -4418.566,E2 -4418.566} C_VEL
LIN {X 0,Y 530.925,Z 603.402,A -85,B 0,C 180,E1 -4419.908,E2 -4419.908} C_VEL
LIN {X 0,Y 531.203,Z 594.484,A -85,B 0,C 180,E1 -4421.059,E2 -4421.059} C_VEL
LIN {X 0,Y 531.488,Z 583.682,A -85,B 0,C 180,E1 -4422.214,E2 -4422.214} C_VEL
LIN {X 0,Y 531.795,Z 572.755,A -85,B 0,C 180,E1 -4423.177,E2 -4423.177} C_VEL
LIN {X 0,Y 532.156,Z 560.801,A -85,B 0,C 180,E1 -4424.043,E2 -4424.043} C_VEL
LIN {X 0,Y 532.521,Z 547.575,A -85,B 0,C 180,E1 -4424.814,E2 -4424.814} C_VEL
LIN {X 0,Y 532.89,Z 534.012,A -85,B 0,C 180,E1 -4425.423,E2 -4425.423} C_VEL
LIN {X 0,Y 533.047,Z 520.38,A -85,B 0,C 180,E1 -4425.878,E2 -4425.878} C_VEL
LIN {X 0,Y 533.297,Z 506.383,A -85,B 0,C 180,E1 -4426.188,E2 -4426.188} C_VEL
LIN {X 0,Y 533.795,Z 381.412,A -85,B 0,C 180,E1 -4427.906,E2 -4427.906} C_VEL
LIN {X 0,Y 531.898,Z 370.61,A -85,B 0,C 180,E1 -4428.125,E2 -4428.125} C_VEL
LIN {X 0,Y 532.44,Z 347.414,A -85,B 0,C 180,E1 -4431.283,E2 -4431.283} C_VEL
LIN {X 0,Y 533.067,Z 323.963,A -85,B 0,C 180,E1 -4434.535,E2 -4434.535} C_VEL
LIN {X 0,Y 532.111,Z 318.051,A -85,B 0,C 180,E1 -4435.419,E2 -4435.419} C_VEL
LIN {X 0,Y 531.009,Z 312.967,A -85,B 0,C 180,E1 -4436.202,E2 -4436.202} C_VEL
LIN {X 0,Y 530.987,Z 312.972,A -85,B 0,C 180,E1 -4439.125,E2 -4439.125} C_VEL
LIN {X 0,Y 530.968,Z 312.966,A -85,B 0,C 180,E1 -4442.1,E2 -4442.1} C_VEL
LIN {X 0,Y 530.987,Z 312.972,A -85,B 0,C 180,E1 -4444.853,E2 -4444.853} C_VEL
LIN {X 0,Y 530.964,Z 312.968,A -85,B 0,C 180,E1 -4447.507,E2 -4447.507} C_VEL
LIN {X 0,Y 530.997,Z 312.967,A -85,B 0,C 180,E1 -4450.43,E2 -4450.43} C_VEL
LIN {X 0,Y 530.96,Z 312.968,A -85,B 0,C 180,E1 -4453.494,E2 -4453.494} C_VEL
LIN {X 0,Y 530.962,Z 312.969,A -85,B 0,C 180,E1 -4456.505,E2 -4456.505} C_VEL
LIN {X 0,Y 530.984,Z 312.965,A -85,B 0,C 180,E1 -4458.975,E2 -4458.975} C_VEL
LIN {X 0,Y 530.953,Z 312.966,A -85,B 0,C 180,E1 -4461.529,E2 -4461.529} C_VEL
LIN {X 0,Y 530.973,Z 312.972,A -85,B 0,C 180,E1 -4464.381,E2 -4464.381} C_VEL
LIN {X 0,Y 530.964,Z 312.966,A -85,B 0,C 180,E1 -4467.133,E2 -4467.133} C_VEL
LIN {X 0,Y 530.98,Z 312.966,A -85,B 0,C 180,E1 -4469.803,E2 -4469.803} C_VEL
LIN {X 0,Y 531.011,Z 312.966,A -85,B 0,C 180,E1 -4472.466,E2 -4472.466} C_VEL
LIN {X 0,Y 530.99,Z 312.964,A -85,B 0,C 180,E1 -4474.941,E2 -4474.941} C_VEL
LIN {X 0,Y 530.963,Z 312.975,A -85,B 0,C 180,E1 -4478.246,E2 -4478.246} C_VEL
LIN {X 0,Y 530.986,Z 312.963,A -85,B 0,C 180,E1 -4480.677,E2 -4480.677} C_VEL
LIN {X 0,Y 530.976,Z 312.965,A -85,B 0,C 180,E1 -4483.07,E2 -4483.07} C_VEL
LIN {X 0,Y 531.01,Z 312.959,A -85,B 0,C 180,E1 -4485.435,E2 -4485.435} C_VEL
LIN {X 0,Y 531.027,Z 312.957,A -85,B 0,C 180,E1 -4488.549,E2 -4488.549} C_VEL
LIN {X 0,Y 531.041,Z 312.962,A -85,B 0,C 180,E1 -4491.629,E2 -4491.629} C_VEL
LIN {X 0,Y 531.104,Z 312.949,A -85,B 0,C 180,E1 -4494.685,E2 -4494.685} C_VEL
LIN {X 0,Y 531.122,Z 312.952,A -85,B 0,C 180,E1 -4497.725,E2 -4497.725} C_VEL
LIN {X 0,Y 531.115,Z 312.951,A -85,B 0,C 180,E1 -4500,E2 -4500} C_VEL
LIN {X 0,Y 531.083,Z 312.953,A -85,B 0,C 180,E1 -4503.034,E2 -4503.034} C_VEL
LIN {X 0,Y 531.022,Z 312.961,A -85,B 0,C 180,E1 -4506.078,E2 -4506.078} C_VEL
LIN {X 0,Y 530.981,Z 312.966,A -85,B 0,C 180,E1 -4509.139,E2 -4509.139} C_VEL
LIN {X 0,Y 531.036,Z 312.962,A -85,B 0,C 180,E1 -4511.669,E2 -4511.669} C_VEL
LIN {X 0,Y 531.007,Z 312.964,A -85,B 0,C 180,E1 -4514.95,E2 -4514.95} C_VEL
LIN {X 0,Y 530.961,Z 312.97,A -85,B 0,C 180,E1 -4517.724,E2 -4517.724} C_VEL
LIN {X 0,Y 531.003,Z 312.962,A -85,B 0,C 180,E1 -4520.128,E2 -4520.128} C_VEL
LIN {X 0,Y 530.929,Z 312.97,A -85,B 0,C 180,E1 -4522.574,E2 -4522.574} C_VEL
LIN {X 0,Y 530.944,Z 312.976,A -85,B 0,C 180,E1 -4525.06,E2 -4525.06} C_VEL
LIN {X 0,Y 530.955,Z 312.967,A -85,B 0,C 180,E1 -4527.598,E2 -4527.598} C_VEL
LIN {X 0,Y 530.951,Z 312.972,A -85,B 0,C 180,E1 -4530.643,E2 -4530.643} C_VEL
LIN {X 0,Y 530.952,Z 312.971,A -85,B 0,C 180,E1 -4533.5,E2 -4533.5} C_VEL
LIN {X 0,Y 530.945,Z 312.973,A -85,B 0,C 180,E1 -4536.559,E2 -4536.559} C_VEL
LIN {X 0,Y 530.975,Z 312.966,A -85,B 0,C 180,E1 -4539.444,E2 -4539.444} C_VEL
LIN {X 0,Y 530.969,Z 312.969,A -85,B 0,C 180,E1 -4542.457,E2 -4542.457} C_VEL
LIN {X 0,Y 530.944,Z 312.97,A -85,B 0,C 180,E1 -4543.519,E2 -4543.519} C_VEL
LIN {X 0,Y 530.269,Z 313.055,A -85,B 0,C 180,E1 -4544.153,E2 -4544.153} C_VEL
LIN {X 0,Y 527.424,Z 313.414,A -85,B 0,C 180,E1 -4545.181,E2 -4545.181} C_VEL
LIN {X 0,Y 525.025,Z 313.717,A -85,B 0,C 180,E1 -4546.01,E2 -4546.01} C_VEL
LIN {X 0,Y 523.993,Z 313.844,A -85,B 0,C 180,E1 -4546.649,E2 -4546.649} C_VEL
LIN {X 0,Y 523.907,Z 313.852,A -85,B 0,C 180,E1 -4546.866,E2 -4546.866} C_VEL
LIN {X 0,Y 523.933,Z 313.848,A -85,B 0,C 180,E1 -4549.87,E2 -4549.87} C_VEL
LIN {X 0,Y 523.966,Z 313.907,A -85,B 0,C 180,E1 -4550.076,E2 -4550.076} C_VEL
LIN {X 0,Y 525.139,Z 320.275,A -85,B 0,C 180,E1 -4551.271,E2 -4551.271} C_VEL
LIN {X 0,Y 524.877,Z 334.011,A -85,B 0,C 180,E1 -4553.669,E2 -4553.669} C_VEL
LIN {X 0,Y 527.218,Z 345.935,A -85,B 0,C 180,E1 -4553.945,E2 -4553.945} C_VEL
LIN {X 0,Y 526.495,Z 470.374,A -85,B 0,C 180,E1 -4555.686,E2 -4555.686} C_VEL
LIN {X 0,Y 526.302,Z 484.317,A -85,B 0,C 180,E1 -4556.031,E2 -4556.031} C_VEL
LIN {X 0,Y 526.046,Z 497.439,A -85,B 0,C 180,E1 -4556.501,E2 -4556.501} C_VEL
LIN {X 0,Y 525.68,Z 510.768,A -85,B 0,C 180,E1 -4557.138,E2 -4557.138} C_VEL
LIN {X 0,Y 525.299,Z 522.856,A -85,B 0,C 180,E1 -4557.873,E2 -4557.873} C_VEL
LIN {X 0,Y 524.886,Z 535.14,A -85,B 0,C 180,E1 -4558.8,E2 -4558.8} C_VEL
LIN {X 0,Y 524.517,Z 546.352,A -85,B 0,C 180,E1 -4559.838,E2 -4559.838} C_VEL
LIN {X 0,Y 524.212,Z 556.458,A -85,B 0,C 180,E1 -4560.974,E2 -4560.974} C_VEL
LIN {X 0,Y 523.911,Z 566.092,A -85,B 0,C 180,E1 -4562.295,E2 -4562.295} C_VEL
LIN {X 0,Y 523.71,Z 573.304,A -85,B 0,C 180,E1 -4563.501,E2 -4563.501} C_VEL
LIN {X 0,Y 523.504,Z 580.443,A -85,B 0,C 180,E1 -4564.984,E2 -4564.984} C_VEL
LIN {X 0,Y 523.463,Z 585.281,A -85,B 0,C 180,E1 -4566.249,E2 -4566.249} C_VEL
LIN {X 0,Y 523.356,Z 588.997,A -85,B 0,C 180,E1 -4567.499,E2 -4567.499} C_VEL
LIN {X 0,Y 523.303,Z 591.726,A -85,B 0,C 180,E1 -4568.74,E2 -4568.74} C_VEL
LIN {X 0,Y 523.289,Z 594,A -85,B 0,C 180,E1 -4570.382,E2 -4570.382} C_VEL
LIN {X 0,Y 523.274,Z 594.78,A -85,B 0,C 180,E1 -4572.007,E2 -4572.007} C_VEL
LIN {X 0,Y 523.238,Z 594.091,A -85,B 0,C 180,E1 -4573.617,E2 -4573.617} C_VEL
LIN {X 0,Y 523.333,Z 591.961,A -85,B 0,C 180,E1 -4575.218,E2 -4575.218} C_VEL
LIN {X 0,Y 523.367,Z 588.401,A -85,B 0,C 180,E1 -4576.805,E2 -4576.805} C_VEL
LIN {X 0,Y 523.486,Z 583.318,A -85,B 0,C 180,E1 -4578.383,E2 -4578.383} C_VEL
LIN {X 0,Y 523.538,Z 578.411,A -85,B 0,C 180,E1 -4579.56,E2 -4579.56} C_VEL
LIN {X 0,Y 523.736,Z 571.356,A -85,B 0,C 180,E1 -4580.929,E2 -4580.929} C_VEL
LIN {X 0,Y 523.989,Z 562.661,A -85,B 0,C 180,E1 -4582.293,E2 -4582.293} C_VEL
LIN {X 0,Y 524.295,Z 553.585,A -85,B 0,C 180,E1 -4583.458,E2 -4583.458} C_VEL
LIN {X 0,Y 524.646,Z 542.629,A -85,B 0,C 180,E1 -4584.62,E2 -4584.62} C_VEL
LIN {X 0,Y 524.979,Z 531.502,A -85,B 0,C 180,E1 -4585.586,E2 -4585.586} C_VEL
LIN {X 0,Y 525.371,Z 519.228,A -85,B 0,C 180,E1 -4586.454,E2 -4586.454} C_VEL
LIN {X 0,Y 525.772,Z 507.398,A -85,B 0,C 180,E1 -4587.127,E2 -4587.127} C_VEL
LIN {X 0,Y 526.079,Z 494.543,A -85,B 0,C 180,E1 -4587.704,E2 -4587.704} C_VEL
LIN {X 0,Y 526.322,Z 480.764,A -85,B 0,C 180,E1 -4588.159,E2 -4588.159} C_VEL
LIN {X 0,Y 526.543,Z 466.303,A -85,B 0,C 180,E1 -4588.471,E2 -4588.471} C_VEL
LIN {X 0,Y 527.098,Z 344.835,A -85,B 0,C 180,E1 -4590.164,E2 -4590.164} C_VEL
LIN {X 0,Y 524.876,Z 333.937,A -85,B 0,C 180,E1 -4590.423,E2 -4590.423} C_VEL
LIN {X 0,Y 525.14,Z 319.856,A -85,B 0,C 180,E1 -4592.877,E2 -4592.877} C_VEL
LIN {X 0,Y 523.93,Z 313.849,A -85,B 0,C 180,E1 -4594.039,E2 -4594.039} C_VEL
LIN {X 0,Y 524.012,Z 313.836,A -85,B 0,C 180,E1 -4596.16,E2 -4596.16} C_VEL
LIN {X 0,Y 523.982,Z 313.839,A -85,B 0,C 180,E1 -4598.485,E2 -4598.485} C_VEL
LIN {X 0,Y 523.995,Z 313.837,A -85,B 0,C 180,E1 -4601.737,E2 -4601.737} C_VEL
LIN {X 0,Y 523.981,Z 313.841,A -85,B 0,C 180,E1 -4605.048,E2 -4605.048} C_VEL
LIN {X 0,Y 523.943,Z 313.841,A -85,B 0,C 180,E1 -4607.97,E2 -4607.97} C_VEL
LIN {X 0,Y 523.955,Z 313.839,A -85,B 0,C 180,E1 -4610.411,E2 -4610.411} C_VEL
LIN {X 0,Y 523.904,Z 313.851,A -85,B 0,C 180,E1 -4612.894,E2 -4612.894} C_VEL
LIN {X 0,Y 523.894,Z 313.85,A -85,B 0,C 180,E1 -4615.422,E2 -4615.422} C_VEL
LIN {X 0,Y 523.895,Z 313.846,A -85,B 0,C 180,E1 -4618.004,E2 -4618.004} C_VEL
LIN {X 0,Y 523.898,Z 313.853,A -85,B 0,C 180,E1 -4620.847,E2 -4620.847} C_VEL
LIN {X 0,Y 523.91,Z 313.845,A -85,B 0,C 180,E1 -4623.727,E2 -4623.727} C_VEL
LIN {X 0,Y 523.858,Z 313.853,A -85,B 0,C 180,E1 -4626.395,E2 -4626.395} C_VEL
LIN {X 0,Y 523.897,Z 313.851,A -85,B 0,C 180,E1 -4629.087,E2 -4629.087} C_VEL
LIN {X 0,Y 523.886,Z 313.848,A -85,B 0,C 180,E1 -4632.126,E2 -4632.126} C_VEL
LIN {X 0,Y 523.927,Z 313.844,A -85,B 0,C 180,E1 -4635.312,E2 -4635.312} C_VEL
LIN {X 0,Y 523.907,Z 313.854,A -85,B 0,C 180,E1 -4638.696,E2 -4638.696} C_VEL
LIN {X 0,Y 523.882,Z 313.848,A -85,B 0,C 180,E1 -4641.896,E2 -4641.896} C_VEL
LIN {X 0,Y 523.912,Z 313.848,A -85,B 0,C 180,E1 -4644.914,E2 -4644.914} C_VEL
LIN {X 0,Y 523.93,Z 313.842,A -85,B 0,C 180,E1 -4647.681,E2 -4647.681} C_VEL
LIN {X 0,Y 523.921,Z 313.849,A -85,B 0,C 180,E1 -4650.684,E2 -4650.684} C_VEL
LIN {X 0,Y 523.899,Z 313.846,A -85,B 0,C 180,E1 -4653.725,E2 -4653.725} C_VEL
LIN {X 0,Y 523.897,Z 313.853,A -85,B 0,C 180,E1 -4656.269,E2 -4656.269} C_VEL
LIN {X 0,Y 523.929,Z 313.845,A -85,B 0,C 180,E1 -4658.766,E2 -4658.766} C_VEL
LIN {X 0,Y 523.929,Z 313.842,A -85,B 0,C 180,E1 -4661.22,E2 -4661.22} C_VEL
LIN {X 0,Y 523.913,Z 313.85,A -85,B 0,C 180,E1 -4664.438,E2 -4664.438} C_VEL
LIN {X 0,Y 523.959,Z 313.84,A -85,B 0,C 180,E1 -4667.608,E2 -4667.608} C_VEL
LIN {X 0,Y 523.937,Z 313.847,A -85,B 0,C 180,E1 -4669.958,E2 -4669.958} C_VEL
LIN {X 0,Y 523.978,Z 313.842,A -85,B 0,C 180,E1 -4672.292,E2 -4672.292} C_VEL
LIN {X 0,Y 524.073,Z 313.826,A -85,B 0,C 180,E1 -4674.614,E2 -4674.614} C_VEL
LIN {X 0,Y 524.111,Z 313.823,A -85,B 0,C 180,E1 -4677.695,E2 -4677.695} C_VEL
LIN {X 0,Y 524.122,Z 313.818,A -85,B 0,C 180,E1 -4680.769,E2 -4680.769} C_VEL
LIN {X 0,Y 524.034,Z 313.829,A -85,B 0,C 180,E1 -4683.075,E2 -4683.075} C_VEL
LIN {X 0,Y 524.028,Z 313.835,A -85,B 0,C 180,E1 -4686.159,E2 -4686.159} C_VEL
LIN {X 0,Y 524.002,Z 313.834,A -85,B 0,C 180,E1 -4688.484,E2 -4688.484} C_VEL
LIN {X 0,Y 524.003,Z 313.841,A -85,B 0,C 180,E1 -4691.738,E2 -4691.738} C_VEL
LIN {X 0,Y 523.997,Z 313.834,A -85,B 0,C 180,E1 -4695.052,E2 -4695.052} C_VEL
LIN {X 0,Y 523.967,Z 313.842,A -85,B 0,C 180,E1 -4697.969,E2 -4697.969} C_VEL
LIN {X 0,Y 523.976,Z 313.837,A -85,B 0,C 180,E1 -4700.41,E2 -4700.41} C_VEL
LIN {X 0,Y 523.914,Z 313.845,A -85,B 0,C 180,E1 -4702.894,E2 -4702.894} C_VEL
LIN {X 0,Y 523.988,Z 313.837,A -85,B 0,C 180,E1 -4706.02,E2 -4706.02} C_VEL
LIN {X 0,Y 523.938,Z 313.842,A -85,B 0,C 180,E1 -4708.875,E2 -4708.875} C_VEL
LIN {X 0,Y 523.925,Z 313.851,A -85,B 0,C 180,E1 -4711.544,E2 -4711.544} C_VEL
LIN {X 0,Y 523.935,Z 313.841,A -85,B 0,C 180,E1 -4714.29,E2 -4714.29} C_VEL
LIN {X 0,Y 523.908,Z 313.85,A -85,B 0,C 180,E1 -4717.132,E2 -4717.132} C_VEL
LIN {X 0,Y 523.941,Z 313.841,A -85,B 0,C 180,E1 -4720.13,E2 -4720.13} C_VEL
LIN {X 0,Y 523.939,Z 313.841,A -85,B 0,C 180,E1 -4722.459,E2 -4722.459} C_VEL
LIN {X 0,Y 523.954,Z 313.847,A -85,B 0,C 180,E1 -4725.309,E2 -4725.309} C_VEL
LIN {X 0,Y 523.959,Z 313.841,A -85,B 0,C 180,E1 -4728.69,E2 -4728.69} C_VEL
LIN {X 0,Y 523.924,Z 313.851,A -85,B 0,C 180,E1 -4731.08,E2 -4731.08} C_VEL
LIN {X 0,Y 523.904,Z 313.846,A -85,B 0,C 180,E1 -4733.825,E2 -4733.825} C_VEL
LIN {X 0,Y 523.945,Z 313.843,A -85,B 0,C 180,E1 -4736.635,E2 -4736.635} C_VEL
LIN {X 0,Y 523.952,Z 313.847,A -85,B 0,C 180,E1 -4739.355,E2 -4739.355} C_VEL
LIN {X 0,Y 523.98,Z 313.843,A -85,B 0,C 180,E1 -4742.281,E2 -4742.281} C_VEL
LIN {X 0,Y 523.993,Z 313.906,A -85,B 0,C 180,E1 -4743.568,E2 -4743.568} C_VEL
LIN {X 0,Y 526.187,Z 324.872,A -85,B 0,C 180,E1 -4745.264,E2 -4745.264} C_VEL
LIN {X 0,Y 525.577,Z 345.805,A -85,B 0,C 180,E1 -4748.218,E2 -4748.218} C_VEL
LIN {X 0,Y 525.07,Z 366.283,A -85,B 0,C 180,E1 -4751.059,E2 -4751.059} C_VEL
LIN {X 0,Y 524.944,Z 370.437,A -85,B 0,C 180,E1 -4751.63,E2 -4751.63} C_VEL
LIN {X 0,Y 527.12,Z 383.241,A -85,B 0,C 180,E1 -4751.887,E2 -4751.887} C_VEL
LIN {X 0,Y 526.452,Z 508.84,A -85,B 0,C 180,E1 -4753.644,E2 -4753.644} C_VEL
LIN {X 0,Y 526.179,Z 523.135,A -85,B 0,C 180,E1 -4753.999,E2 -4753.999} C_VEL
LIN {X 0,Y 525.9,Z 536.841,A -85,B 0,C 180,E1 -4754.497,E2 -4754.497} C_VEL
LIN {X 0,Y 525.561,Z 549.077,A -85,B 0,C 180,E1 -4755.082,E2 -4755.082} C_VEL
LIN {X 0,Y 525.179,Z 561.95,A -85,B 0,C 180,E1 -4755.863,E2 -4755.863} C_VEL
LIN {X 0,Y 524.796,Z 573.657,A -85,B 0,C 180,E1 -4756.741,E2 -4756.741} C_VEL
LIN {X 0,Y 524.445,Z 584.519,A -85,B 0,C 180,E1 -4757.73,E2 -4757.73} C_VEL
LIN {X 0,Y 524.175,Z 594.205,A -85,B 0,C 180,E1 -4758.789,E2 -4758.789} C_VEL
LIN {X 0,Y 523.874,Z 603.124,A -85,B 0,C 180,E1 -4759.956,E2 -4759.956} C_VEL
LIN {X 0,Y 523.726,Z 610.551,A -85,B 0,C 180,E1 -4761.122,E2 -4761.122} C_VEL
LIN {X 0,Y 523.57,Z 616.743,A -85,B 0,C 180,E1 -4762.285,E2 -4762.285} C_VEL
LIN {X 0,Y 523.457,Z 623.32,A -85,B 0,C 180,E1 -4763.833,E2 -4763.833} C_VEL
LIN {X 0,Y 523.377,Z 627.169,A -85,B 0,C 180,E1 -4764.992,E2 -4764.992} C_VEL
LIN {X 0,Y 523.419,Z 630.137,A -85,B 0,C 180,E1 -4766.15,E2 -4766.15} C_VEL
LIN {X 0,Y 523.333,Z 632.85,A -85,B 0,C 180,E1 -4767.69,E2 -4767.69} C_VEL
LIN {X 0,Y 523.247,Z 634.193,A -85,B 0,C 180,E1 -4769.23,E2 -4769.23} C_VEL
LIN {X 0,Y 523.247,Z 634.194,A -85,B 0,C 180,E1 -4770.769,E2 -4770.769} C_VEL
LIN {X 0,Y 523.333,Z 632.854,A -85,B 0,C 180,E1 -4772.308,E2 -4772.308} C_VEL
LIN {X 0,Y 523.419,Z 630.142,A -85,B 0,C 180,E1 -4773.849,E2 -4773.849} C_VEL
LIN {X 0,Y 523.452,Z 625.98,A -85,B 0,C 180,E1 -4775.392,E2 -4775.392} C_VEL
LIN {X 0,Y 523.494,Z 620.245,A -85,B 0,C 180,E1 -4776.939,E2 -4776.939} C_VEL
LIN {X 0,Y 523.634,Z 613.785,A -85,B 0,C 180,E1 -4778.295,E2 -4778.295} C_VEL
LIN {X 0,Y 523.814,Z 605.758,A -85,B 0,C 180,E1 -4779.654,E2 -4779.654} C_VEL
LIN {X 0,Y 524.105,Z 597.367,A -85,B 0,C 180,E1 -4780.82,E2 -4780.82} C_VEL
LIN {X 0,Y 524.418,Z 586.596,A -85,B 0,C 180,E1 -4782.06,E2 -4782.06} C_VEL
LIN {X 0,Y 524.716,Z 575.997,A -85,B 0,C 180,E1 -4783.062,E2 -4783.062} C_VEL
LIN {X 0,Y 525.059,Z 564.795,A -85,B 0,C 180,E1 -4783.941,E2 -4783.941} C_VEL
LIN {X 0,Y 525.454,Z 552.601,A -85,B 0,C 180,E1 -4784.721,E2 -4784.721} C_VEL
LIN {X 0,Y 525.815,Z 539.072,A -85,B 0,C 180,E1 -4785.405,E2 -4785.405} C_VEL
LIN {X 0,Y 526.09,Z 525.444,A -85,B 0,C 180,E1 -4785.926,E2 -4785.926} C_VEL
LIN {X 0,Y 526.391,Z 511.109,A -85,B 0,C 180,E1 -4786.307,E2 -4786.307} C_VEL
LIN {X 0,Y 526.552,Z 490.73,A -85,B 0,C 180,E1 -4786.626,E2 -4786.626} C_VEL
LIN {X 0,Y 527.131,Z 383.169,A -85,B 0,C 180,E1 -4788.112,E2 -4788.112} C_VEL
LIN {X 0,Y 524.928,Z 370.247,A -85,B 0,C 180,E1 -4788.384,E2 -4788.384} C_VEL
LIN {X 0,Y 525.512,Z 348.605,A -85,B 0,C 180,E1 -4791.372,E2 -4791.372} C_VEL
LIN {X 0,Y 526.123,Z 326.637,A -85,B 0,C 180,E1 -4794.462,E2 -4794.462} C_VEL
LIN {X 0,Y 525.961,Z 323.206,A -85,B 0,C 180,E1 -4794.963,E2 -4794.963} C_VEL
LIN {X 0,Y 523.958,Z 313.845,A -85,B 0,C 180,E1 -4796.432,E2 -4796.432} C_VEL
LIN {X 0,Y 523.953,Z 313.846,A -85,B 0,C 180,E1 -4799.323,E2 -4799.323} C_VEL
LIN {X 0,Y 523.934,Z 313.845,A -85,B 0,C 180,E1 -4802.448,E2 -4802.448} C_VEL
LIN {X 0,Y 523.933,Z 313.846,A -85,B 0,C 180,E1 -4805.224,E2 -4805.224} C_VEL
LIN {X 0,Y 523.914,Z 313.846,A -85,B 0,C 180,E1 -4808.101,E2 -4808.101} C_VEL
LIN {X 0,Y 523.957,Z 313.841,A -85,B 0,C 180,E1 -4811.089,E2 -4811.089} C_VEL
LIN {X 0,Y 523.937,Z 313.846,A -85,B 0,C 180,E1 -4814.227,E2 -4814.227} C_VEL
LIN {X 0,Y 523.921,Z 313.85,A -85,B 0,C 180,E1 -4816.833,E2 -4816.833} C_VEL
LIN {X 0,Y 523.94,Z 313.843,A -85,B 0,C 180,E1 -4818.907,E2 -4818.907} C_VEL
LIN {X 0,Y 523.911,Z 313.844,A -85,B 0,C 180,E1 -4821.898,E2 -4821.898} C_VEL
LIN {X 0,Y 523.93,Z 313.846,A -85,B 0,C 180,E1 -4824.909,E2 -4824.909} C_VEL
LIN {X 0,Y 523.931,Z 313.842,A -85,B 0,C 180,E1 -4827.678,E2 -4827.678} C_VEL
LIN {X 0,Y 523.963,Z 313.842,A -85,B 0,C 180,E1 -4830.673,E2 -4830.673} C_VEL
LIN {X 0,Y 523.971,Z 313.838,A -85,B 0,C 180,E1 -4833.728,E2 -4833.728} C_VEL
LIN {X 0,Y 523.905,Z 313.852,A -85,B 0,C 180,E1 -4836.269,E2 -4836.269} C_VEL
LIN {X 0,Y 523.938,Z 313.843,A -85,B 0,C 180,E1 -4838.766,E2 -4838.766} C_VEL
LIN {X 0,Y 523.943,Z 313.838,A -85,B 0,C 180,E1 -4841.22,E2 -4841.22} C_VEL
LIN {X 0,Y 523.927,Z 313.846,A -85,B 0,C 180,E1 -4843.638,E2 -4843.638} C_VEL
LIN {X 0,Y 523.93,Z 313.849,A -85,B 0,C 180,E1 -4846.028,E2 -4846.028} C_VEL
LIN {X 0,Y 524.004,Z 313.833,A -85,B 0,C 180,E1 -4848.394,E2 -4848.394} C_VEL
LIN {X 0,Y 523.989,Z 313.839,A -85,B 0,C 180,E1 -4851.516,E2 -4851.516} C_VEL
LIN {X 0,Y 524.065,Z 313.826,A -85,B 0,C 180,E1 -4854.613,E2 -4854.613} C_VEL
LIN {X 0,Y 524.095,Z 313.827,A -85,B 0,C 180,E1 -4857.694,E2 -4857.694} C_VEL
LIN {X 0,Y 524.084,Z 313.827,A -85,B 0,C 180,E1 -4860,E2 -4860} C_VEL
LIN {X 0,Y 524.024,Z 313.832,A -85,B 0,C 180,E1 -4863.075,E2 -4863.075} C_VEL
LIN {X 0,Y 523.985,Z 313.837,A -85,B 0,C 180,E1 -4866.159,E2 -4866.159} C_VEL
LIN {X 0,Y 523.934,Z 313.846,A -85,B 0,C 180,E1 -4869.263,E2 -4869.263} C_VEL
LIN {X 0,Y 523.984,Z 313.839,A -85,B 0,C 180,E1 -4871.734,E2 -4871.734} C_VEL
LIN {X 0,Y 523.971,Z 313.841,A -85,B 0,C 180,E1 -4875.047,E2 -4875.047} C_VEL
LIN {X 0,Y 523.903,Z 313.847,A -85,B 0,C 180,E1 -4877.971,E2 -4877.971} C_VEL
LIN {X 0,Y 523.94,Z 313.841,A -85,B 0,C 180,E1 -4880.411,E2 -4880.411} C_VEL
LIN {X 0,Y 523.895,Z 313.849,A -85,B 0,C 180,E1 -4882.894,E2 -4882.894} C_VEL
